DATA_BLOCK "DB2040_WINCC_HMI_LINES"   // DB2040
{ S7_Optimized_Access := 'FALSE'; DB_Accessible_From_OPC_UA := 'FALSE' }
AUTHOR : ETXETAR
VERSION : 1.0
// stored: AutoNumber false, DBAccessibleFromOPCUA false, DBAccessibleFromWebserver true, IsOnlyStoredInLoadMemory false, IsWriteProtectedInAS false
   VAR RETAIN
      MODES { S7_SetPoint := 'True'} : Array[1..5] of "WINCC_HMI_LINES";
      SERVICES { S7_SetPoint := 'True'} : Array[1..30] of "WINCC_HMI_LINES";
   END_VAR
BEGIN
   // MODES[1] : AUTOMATIC MODE
   // MODES[2] : SEMIAUTO MODE
   // MODES[3] : MANUAL MODE
   // MODES[1].WINCC_LINE_REQUEST_RIGHT : AUTOMATIC MODE RIGHT REQUEST
   // MODES[2].WINCC_LINE_REQUEST_RIGHT : SEMIAUTO MODE RIGHT REQUEST
   // MODES[3].WINCC_LINE_REQUEST_RIGHT : MANUAL MODE RIGHT REQUEST
   // MODES[1].WINCC_LINE_REQUEST_LEFT : AUTOMATIC MODE LEFT REQUEST
   // MODES[2].WINCC_LINE_REQUEST_LEFT : SEMIAUTO MODE LEFT REQUEST
   // MODES[3].WINCC_LINE_REQUEST_LEFT : MANUAL MODE LEFT REQUEST
   // MODES[1].WINCC_LINE_CONDITIONS_RIGHT : AUTOMATIC MODE RIGHT CONDITIONS
   // MODES[2].WINCC_LINE_CONDITIONS_RIGHT : SEMIAUTO MODE RIGHT CONDITIONS
   // MODES[3].WINCC_LINE_CONDITIONS_RIGHT : MANUAL MODE RIGHT CONDITIONS
   // MODES[1].WINCC_LINE_CONDITIONS_LEFT : AUTOMATIC MODE LEFT CONDITIONS
   // MODES[2].WINCC_LINE_CONDITIONS_LEFT : SEMIAUTO MODE LEFT CONDITIONS
   // MODES[3].WINCC_LINE_CONDITIONS_LEFT : MANUAL MODE LEFT CONDITIONS
   // MODES[1].WINCC_LINE_ACTIVE_RIGHT : AUTOMATIC MODE RIGHT ACTIVE
   // MODES[2].WINCC_LINE_ACTIVE_RIGHT : SEMIAUTO MODE RIGHT ACTIVE
   // MODES[3].WINCC_LINE_ACTIVE_RIGHT : MANUAL MODE RIGHT ACTIVE
   // MODES[1].WINCC_LINE_ACTIVE_LEFT : AUTOMATIC MODE LEFT ACTIVE
   // MODES[2].WINCC_LINE_ACTIVE_LEFT : SEMIAUTO MODE LEFT ACTIVE
   // MODES[3].WINCC_LINE_ACTIVE_LEFT : MANUAL MODE LEFT ACTIVE
   // MODES[1].WINCC_LINE_STATUS_1_RIGHT : AUTOMATIC MODE RIGHT STATUS
   // MODES[2].WINCC_LINE_STATUS_1_RIGHT : SEMIAUTO MODE RIGHT STATUS
   // MODES[3].WINCC_LINE_STATUS_1_RIGHT : MANUAL MODE RIGHT STATUS
   // MODES[1].WINCC_LINE_STATUS_1_LEFT : AUTOMATIC MODE LEFT STATUS
   // MODES[2].WINCC_LINE_STATUS_1_LEFT : SEMIAUTO MODE LEFT STATUS
   // MODES[3].WINCC_LINE_STATUS_1_LEFT : MANUAL MODE LEFT STATUS
   // SERVICES[1] : PNEUMATIC SYSTEM
   // SERVICES[2] : POWDER FEEDER 1 GENERAL UNIT 01
   // SERVICES[3] : POWDER FEEDER 1 GENERAL UNIT 02
   // SERVICES[4] : POWDER FEEDER 2 GENERAL UNIT 02
   // SERVICES[5] : POWDER FEEDER 1 HEATER JKL UNIT 01 LINE 1
   // SERVICES[6] : POWDER FEEDER 1 HEATER JKL UNIT 01 LINE 2
   // SERVICES[7] : POWDER FEEDER 1 HEATER JKL UNIT 02 LINE 1
   // SERVICES[8] : POWDER FEEDER 1 HEATER JKL UNIT 02 LINE 2
   // SERVICES[9] : POWDER FEEDER 2 HEATER JKL UNIT 02 LINE 1
   // SERVICES[10] : POWDER FEEDER 1 HOPPER UNIT 01 LINE 1
   // SERVICES[11] : POWDER FEEDER 1 HOPPER UNIT 01 LINE 2
   // SERVICES[12] : POWDER FEEDER 1 HOPPER UNIT 02 LINE 1
   // SERVICES[13] : POWDER FEEDER 1 HOPPER UNIT 02 LINE 2
   // SERVICES[14] : POWDER FEEDER 2 HOPPER UNIT 02 LINE 1
END_DATA_BLOCK

DATA_BLOCK "DB2041_WINCC_HMI_LINES_STATIONS"   // DB2041
{ S7_Optimized_Access := 'FALSE'; DB_Accessible_From_OPC_UA := 'FALSE' }
AUTHOR : ETXETAR
VERSION : 1.0
// stored: AutoNumber false, DBAccessibleFromOPCUA false, DBAccessibleFromWebserver true, IsOnlyStoredInLoadMemory false, IsWriteProtectedInAS false
   VAR RETAIN
      STATION_1 { S7_SetPoint := 'True'} : Array[1..20] of "WINCC_HMI_LINES";
      STATION_2 { S7_SetPoint := 'True'} : Array[1..20] of "WINCC_HMI_LINES";
      STATION_3 { S7_SetPoint := 'True'} : Array[1..20] of "WINCC_HMI_LINES";
      STATION_4 { S7_SetPoint := 'True'} : Array[1..20] of "WINCC_HMI_LINES";
      STATION_5 { S7_SetPoint := 'True'} : Array[1..20] of "WINCC_HMI_LINES";
      STATION_6 { S7_SetPoint := 'True'} : Array[1..20] of "WINCC_HMI_LINES";
      STATION_7 { S7_SetPoint := 'True'} : Array[1..20] of "WINCC_HMI_LINES";
      STATION_8 { S7_SetPoint := 'True'} : Array[1..20] of "WINCC_HMI_LINES";
      STATION_9 { S7_SetPoint := 'True'} : Array[1..20] of "WINCC_HMI_LINES";
      STATION_10 { S7_SetPoint := 'True'} : Array[1..20] of "WINCC_HMI_LINES";
   END_VAR
BEGIN
END_DATA_BLOCK

DATA_BLOCK "DB2050_HARDWARE_SOFTWARE_ENABLE_DISABLE"   // DB2050
{ S7_Optimized_Access := 'FALSE'; DB_Accessible_From_OPC_UA := 'FALSE' }
AUTHOR : ETXETAR
VERSION : 1.0
// stored: AutoNumber false, DBAccessibleFromOPCUA false, DBAccessibleFromWebserver true, IsOnlyStoredInLoadMemory false, IsWriteProtectedInAS false
   VAR RETAIN
      DISABLE_PART : Struct
         HW_GENERAL_CONDITIONS : Bool;   // HARDWARE GENERAL CONDITIONS
         SW_GENERAL_CONDITIONS : Bool;   // SOFTWARE GENERAL CONDITIONS
         PART_A_ENABLE : Bool;   // PART A ENABLE
         PART_B_ENABLE : Bool;   // PART B ENABLE
         PART_C_ENABLE : Bool;   // PART C ENABLE
         PART_D_ENABLE : Bool;   // PART D ENABLE
         PART_E_ENABLE : Bool;   // PART E ENABLE
         PART_F_ENABLE : Bool;   // PART F ENABLE
         HW_PART_A_ENABLE_REQUEST : Bool;   // HARDWARE PART A ENABLE REQUEST
         HW_PART_A_DISABLE_REQUEST : Bool;   // HARDWARE PART A DISABLE REQUEST
         HW_PART_B_ENABLE_REQUEST : Bool;   // HARDWARE PART B ENABLE REQUEST
         HW_PART_B_DISABLE_REQUEST : Bool;   // HARDWARE PART B DISABLE REQUEST
         HW_PART_C_ENABLE_REQUEST : Bool;   // HARDWARE PART C ENABLE REQUEST
         HW_PART_C_DISABLE_REQUEST : Bool;   // HARDWARE PART C DISABLE REQUEST
         HW_PART_D_ENABLE_REQUEST : Bool;   // HARDWARE PART D ENABLE REQUEST
         HW_PART_D_DISABLE_REQUEST : Bool;   // HARDWARE PART D DISABLE REQUEST
         HW_PART_E_ENABLE_REQUEST : Bool;   // HARDWARE PART E ENABLE REQUEST
         HW_PART_E_DISABLE_REQUEST : Bool;   // HARDWARE PART E DISABLE REQUEST
         HW_PART_F_ENABLE_REQUEST : Bool;   // HARDWARE PART F ENABLE REQUEST
         HW_PART_F_DISABLE_REQUEST : Bool;   // HARDWARE PART F DISABLE REQUEST
         HW_PART_ENABLE_DISABLE_REQUEST : Bool;   // HARDWARE ENABLE DISABLE REQUEST
         SW_PART_A_ENABLE_REQUEST : Bool;   // SOFTWARE PART A ENABLE REQUEST
         SW_PART_A_DISABLE_REQUEST : Bool;   // SOFTWARE PART A DISABLE REQUEST
         SW_PART_B_ENABLE_REQUEST : Bool;   // SOFTWARE PART B ENABLE REQUEST
         SW_PART_B_DISABLE_REQUEST : Bool;   // SOFTWARE PART B DISABLE REQUEST
         SW_PART_C_ENABLE_REQUEST : Bool;   // SOFTWARE PART C ENABLE REQUEST
         SW_PART_C_DISABLE_REQUEST : Bool;   // SOFTWARE PART C DISABLE REQUEST
         SW_PART_D_ENABLE_REQUEST : Bool;   // SOFTWARE PART D ENABLE REQUEST
         SW_PART_D_DISABLE_REQUEST : Bool;   // SOFTWARE PART D DISABLE REQUEST
         SW_PART_E_ENABLE_REQUEST : Bool;   // SOFTWARE PART E ENABLE REQUEST
         SW_PART_E_DISABLE_REQUEST : Bool;   // SOFTWARE PART E DISABLE REQUEST
         SW_PART_F_ENABLE_REQUEST : Bool;   // SOFTWARE PART F ENABLE REQUEST
         SW_PART_F_DISABLE_REQUEST : Bool;   // SOFTWARE PART F DISABLE REQUEST
         SW_PART_ENABLE_DISABLE_REQUEST : Bool;   // SOFTWARE ENABLE DISABLE REQUEST
         HMI_ACCEPT_BUTTON : Bool;   // HMI ACCEPT BUTTON
         HW_PART_A_ENABLED : Bool := true;   // HARDWARE PART A ENABLED
         HW_PART_B_ENABLED : Bool := true;   // HARDWARE PART B ENABLED
         HW_PART_C_ENABLED : Bool := true;   // HARDWARE PART C ENABLED
         HW_PART_D_ENABLED : Bool;   // HARDWARE PART D ENABLED
         HW_PART_E_ENABLED : Bool;   // HARDWARE PART E ENABLED
         HW_PART_F_ENABLED : Bool;   // HARDWARE PART F ENABLED
         SW_PART_A_ENABLED : Bool := true;   // SOFTWARE PART A ENABLED
         SW_PART_B_ENABLED : Bool := true;   // SOFTWARE PART B ENABLED
         SW_PART_C_ENABLED : Bool := true;   // SOFTWARE PART C ENABLED
         SW_PART_D_ENABLED : Bool;   // SOFTWARE PART D ENABLED
         SW_PART_E_ENABLED : Bool;   // SOFTWARE PART E ENABLED
         SW_PART_F_ENABLED : Bool;   // SOFTWARE PART F ENABLED
         PART_A_DISABLE_ALARM : Bool;   // PART A DISABLE ALARM
         PART_B_DISABLE_ALARM : Bool;   // PART B DISABLE ALARM
         PART_C_DISABLE_ALARM : Bool;   // PART C DISABLE ALARM
         PART_D_DISABLE_ALARM : Bool;   // PART D DISABLE ALARM
         PART_E_DISABLE_ALARM : Bool;   // PART E DISABLE ALARM
         PART_F_DISABLE_ALARM : Bool;   // PART F DISABLE ALARM
         DESELECT_IN_PROGRESS : Bool;   // DESELECTION IN PROGRESS
         HW_DISABLED_ACK : Bool;   // HARDWARE DISABLED ACKNOWLEDGE
         HW_DISABLED_ACK_AUX : Bool;   // HARDWARE DISABLED ACKNOWLEDGE AUXILIARY
         ALL_HW_PARTS_DISABLED : Bool;   // ALL HARDWARE PARTS DISABLED
         ALL_SW_PARTS_DISABLED : Bool;   // ALL SOFTWARE PARTS DISABLED
         ALL_HARDWARE_ENABLED : Bool;   // ALL HARDWARE ENABLED
         PART_A_DISABLED_SCRIPT_COMMAND : Bool;   // PART A DISABLED SCRIPT COMMAND
         PART_A_ENABLED_SCRIPT_COMMAND : Bool;   // PART A ENABLED SCRIPT COMMAND
         PART_B_DISABLED_SCRIPT_COMMAND : Bool;   // PART B DISABLED SCRIPT COMMAND
         PART_B_ENABLED_SCRIPT_COMMAND : Bool;   // PART B ENABLED SCRIPT COMMAND
         PART_C_DISABLED_SCRIPT_COMMAND : Bool;   // PART C DISABLED SCRIPT COMMAND
         PART_C_ENABLED_SCRIPT_COMMAND : Bool;   // PART C ENABLED SCRIPT COMMAND
         PART_D_DISABLED_SCRIPT_COMMAND : Bool;   // PART D DISABLED SCRIPT COMMAND
         PART_D_ENABLED_SCRIPT_COMMAND : Bool;   // PART D ENABLED SCRIPT COMMAND
         PART_E_DISABLED_SCRIPT_COMMAND : Bool;   // PART E DISABLED SCRIPT COMMAND
         PART_E_ENABLED_SCRIPT_COMMAND : Bool;   // PART E ENABLED SCRIPT COMMAND
         PART_F_DISABLED_SCRIPT_COMMAND : Bool;   // PART F DISABLED SCRIPT COMMAND
         PART_F_ENABLED_SCRIPT_COMMAND : Bool;   // PART F ENABLED SCRIPT COMMAND
         ALARM_SCREEN : Int;   // HMI ALARMS SCREEN NUMBER
         ENABLE_MACHINE_STRUCTURE_SCREEN : Int;   // HMI ENABLE MACHINE STRUCTURE SCREEN NUMBER
         SW_PULSE : Array[1..16] of Bool;
         HW_PULSE : Array[1..16] of Bool;
      END_STRUCT;
   END_VAR
BEGIN
END_DATA_BLOCK

DATA_BLOCK "DB21000_POWDER_FEEDER_GENERAL"   // DB21000
{ S7_Optimized_Access := 'FALSE'; DB_Accessible_From_OPC_UA := 'FALSE' }
VERSION : 0.1
// stored: AutoNumber false, DBAccessibleFromOPCUA false, DBAccessibleFromWebserver true, IsOnlyStoredInLoadMemory false, IsWriteProtectedInAS false
   VAR
      POWDER_FEEDER_1_UNIT_01 : "POWDER FEEDER GENERAL";
      POWDER_FEEDER_1_UNIT_02 { S7_SetPoint := 'True'} : "POWDER FEEDER GENERAL";
      POWDER_FEEDER_2_UNIT_02 { S7_SetPoint := 'True'} : "POWDER FEEDER GENERAL";
   END_VAR
BEGIN
END_DATA_BLOCK

DATA_BLOCK "DB21002_POWDER_FEEDER_OERLIKON_INTERLOCK"   // DB21002
{ S7_Optimized_Access := 'FALSE'; DB_Accessible_From_OPC_UA := 'FALSE' }
VERSION : 0.1
// stored: AutoNumber false, DBAccessibleFromOPCUA false, DBAccessibleFromWebserver true, IsOnlyStoredInLoadMemory false, IsWriteProtectedInAS false
   VAR
      POWDER_FEEDER_1_UNIT_01 : "POWDER FEEDER OERLIKON";
      POWDER_FEEDER_1_UNIT_02 : "POWDER FEEDER OERLIKON";
      POWDER_FEEDER_2_UNIT_02 : "POWDER FEEDER OERLIKON";
   END_VAR
BEGIN
END_DATA_BLOCK

DATA_BLOCK "DB21003_POWDER_FEEDER_HMI_INTERLOCK"   // DB21003
{ S7_Optimized_Access := 'FALSE'; DB_Accessible_From_OPC_UA := 'FALSE' }
VERSION : 0.1
// stored: AutoNumber false, DBAccessibleFromOPCUA false, DBAccessibleFromWebserver true, IsOnlyStoredInLoadMemory false, IsWriteProtectedInAS false
   VAR
      POWDER_FEEDER_1_UNIT_01 : Struct
         "HMI_Values Setpoints" : "POWDER FEEDER HMI VALUES SETPOINTS";
         "HMI_Offsets Alarms and Warnings" : "POWDER FEEDER HMI OFFSETS ALARMS WARNINGS";
         HMI_ACTIONS_STATUS { S7_SetPoint := 'True'} : "POWDER FEEDER HMI ACTIONS";
      END_STRUCT;
      POWDER_FEEDER_1_UNIT_02 : Struct
         "HMI_Values Setpoints" : "POWDER FEEDER HMI VALUES SETPOINTS";
         "HMI_Offsets Alarms and Warnings" : "POWDER FEEDER HMI OFFSETS ALARMS WARNINGS";
         HMI_ACTIONS_STATUS : "POWDER FEEDER HMI ACTIONS";
      END_STRUCT;
      POWDER_FEEDER_2_UNIT_02 : Struct
         "HMI_Values Setpoints" : "POWDER FEEDER HMI VALUES SETPOINTS";
         "HMI_Offsets Alarms and Warnings" : "POWDER FEEDER HMI OFFSETS ALARMS WARNINGS";
         HMI_ACTIONS_STATUS : "POWDER FEEDER HMI ACTIONS";
      END_STRUCT;
   END_VAR
BEGIN
END_DATA_BLOCK

DATA_BLOCK "DB21004_POWDER_FEEDER_CNC_INTERLOCK"   // DB21004
{ S7_Optimized_Access := 'FALSE'; DB_Accessible_From_OPC_UA := 'FALSE' }
VERSION : 0.1
// stored: AutoNumber false, DBAccessibleFromOPCUA false, DBAccessibleFromWebserver true, IsOnlyStoredInLoadMemory false, IsWriteProtectedInAS false
   VAR
      POWDER_FEEDER_1_UNIT_01 : "POWDER FEEDER CNC VALUES SETPOINTS";
      POWDER_FEEDER_1_UNIT_02 : "POWDER FEEDER CNC VALUES SETPOINTS";
      POWDER_FEEDER_2_UNIT_02 : "POWDER FEEDER CNC VALUES SETPOINTS";
   END_VAR
BEGIN
END_DATA_BLOCK

DATA_BLOCK "DB21005_POWDER_FEEDER_PLC_AUX"   // DB21005
{ S7_Optimized_Access := 'FALSE'; DB_Accessible_From_OPC_UA := 'FALSE' }
VERSION : 0.1
// stored: AutoNumber false, DBAccessibleFromOPCUA false, DBAccessibleFromWebserver true, IsOnlyStoredInLoadMemory false, IsWriteProtectedInAS false
   VAR
      "INTERLOCKS_PLC_I/O_PF_1_UNIT_01" : "POWDER FEEDER PLC AUXILIAR";
      "INTERLOCKS_PLC_I/O_PF_1_UNIT_02" : "POWDER FEEDER PLC AUXILIAR";
      "INTERLOCKS_PLC_I/O_PF_2_UNIT_02" : "POWDER FEEDER PLC AUXILIAR";
   END_VAR
BEGIN
END_DATA_BLOCK

DATA_BLOCK "DB1101_MACHINE_SEQUENCE"   // DB1101
{ S7_Optimized_Access := 'FALSE'; DB_Accessible_From_OPC_UA := 'FALSE' }
AUTHOR : ETXETAR
VERSION : 1.0
// stored: AutoNumber false, DBAccessibleFromOPCUA false, DBAccessibleFromWebserver true, IsOnlyStoredInLoadMemory false, IsWriteProtectedInAS false
   VAR RETAIN
      GENERAL_CONDITIONS : Bool;   // MACHINING SEQUENCE GENERAL CONDITIONS / MACHINE SEQUENCE GENERAL CONDITIONS
      INITIAL_CONDITIONS : Bool;   // MACHINING SEQUENCE INITIAL CONDITIONS / MACHINE SEQUENCE INITIAL CONDITIONS
      START_REQUEST : Bool;   // MACHINING SEQUENCE START REQUEST / MACHINE SEQUENCE START REQUEST
      COMMAND : Bool;   // MACHINING SEQUENCE COMMAND / MACHINE SEQUENCE COMMAND
      REQUEST : Bool;   // MACHINING SEQUENCE REQUEST DELAYED / MACHINE SEQUENCE REQUEST
      COMMAND_PULSE : Bool;   // MACHINING SEQUENCE COMMAND PULSE / MACHINE SEQUENCE COMMAND PULSE
      REQUEST_PULSE : Bool;   // MACHINING SEQUENCE REQUEST PULSE / MACHINE SEQUENCE REQUEST PULSE
      RUNNING : Bool;   // MACHINING SEQUENCE IN PROCESS / MACHINE SEQUENCE RUNNING
      CYCLE_UNIT_01 : Bool;   // MACHINING SEQUENCE CYCLE STATION 01R / MACHINE SEQUENCE CYCLE UNIT 01
      CYCLE_UNIT_02 : Bool;   // MACHINING SEQUENCE CYCLE STATION 01L / MACHINE SEQUENCE CYCLE UNIT 02
      CYCLE_UNIT_03 : Bool;   // MACHINING SEQUENCE CYCLE STATION 01L / MACHINE SEQUENCE CYCLE UNIT 03
      NO_PART_AT_FEED_UNIT_01 : Bool;   // MACHINING SEQUENCE CYCLE STATION FIXTURE / MACHINE SEQUENCE NO PART AT FEED UNIT 02
      DELIVERY_OCCUPIED_UNIT_01 : Bool;   // MACHINING SEQUENCE CYCLE PART HANDLING DEVICE / MACHINE SEQUENCE DELIVERY OCCUPIED UNIT 02
      NO_PART_AT_FEED_UNIT_02 : Bool;   // MACHINING SEQUENCE NO PART AT FEED / MACHINE SEQUENCE NO PART AT FEED UNIT 02
      DELIVERY_OCCUPIED_UNIT_02 : Bool;   // MACHINING SEQUENCE DELIVERY OCCUPIED / MACHINE SEQUENCE DELIVERY OCCUPIED UNIT 02
      CLEAR_TO_LOAD_UNLOAD_UNIT_01 : Bool;   // MACHINING SEQUENCE OUT OF COLLISION TO PART HANDLING DEVICE / MACHINE SEQUENCE CLEAR TO LOAD UNLOAD MACHINE UNIT 01
      CLEAR_TO_LOAD_UNLOAD_UNIT_02 : Bool;   // MACHINING SEQUENCE OUT OF COLLISION TO PART HANDLING DEVICE / MACHINE SEQUENCE CLEAR TO LOAD UNLOAD MACHINE UNIT 02
      SKIP_FIXTURE_UNIT_01 : Bool;   // MACHINING SEQUENCE CLAMP FIXTURE 1 / MACHINE SEQUENCE SKIP FIXTURE UNIT 01
      SKIP_FIXTURE_UNIT_02 : Bool;   // MACHINING SEQUENCE CLAMP FIXTURE 2 / MACHINE SEQUENCE SKIP FIXTURE UNIT 02
      SPARE_1 : Bool;   // MACHINING SEQUENCE UNCLAMP FIXTURE 1 / MACHINE SEQUENCE
      SPARE_2 : Bool;   // MACHINING SEQUENCE UNCLAMP FIXTURE 2 / MACHINE SEQUENCE
      RESET_PLC_AND_CNC : Bool;   // MACHINING SEQUENCE RESET PLC AND CNC / MACHINE SEQUENCE RESET PLC AND CNC
      FULL_DEPTH : Bool;   // MACHINING SEQUENCE FULL DEPTH / MACHINE SEQUENCE FULL DEPTH
      TIME_EXCEEDED : Bool;   // MACHINING SEQUENCE TIME EXCEEDED / MACHINE SEQUENCE TIME EXCEEDED
      PREALARM : Bool;   // MACHINING SEQUENCE PREALARM / MACHINE SEQUENCE PREALARM
      LOADER_CHECK_PART_READY : Bool;   // MACHINING SEQUENCE LOADER CHECK PART READY / MACHINE SEQUENCE LOADER CHECK PART READY
      LOADER_RESET_CHECK_PART_READY : Bool;   // MACHINING SEQUENCE RST LOADER CHECK PART READY / MACHINE SEQUENCE LOADER RESET CHECK PART READY
      PREALARM_GONE : Bool;   // MACHINING SEQUENCE PREALARM GONE / MACHINE SEQUENCE PREALARM GONE
      AUX1 : Bool;   // MACHINING SEQUENCE AUX1 / MACHINE SEQUENCE AUX1
      AUX2 : Bool;   // MACHINING SEQUENCE AUX2 / MACHINE SEQUENCE AUX2
      AUX3 : Bool;   // MACHINING SEQUENCE AUX3 / MACHINE SEQUENCE AUX3
      START_GENERAL_COND_HELP : Bool;   // MACHINING SEQUENCE START GENERAL CONDITIONS HELP / MACHINE SEQUENCE START GENERAL COND HELP
      START_INITIAL_COND_HELP : Bool;   // MACHINING SEQUENCE START INITIAL CONDITIONS HELP / MACHINE SEQUENCE START INITIAL COND HELP
      TIMER_MACHINE_START_REQUEST : TON_TIME;   // MACHINE SEQUENCE START REQUEST TIMER
      "TIMER_TIME _EXCEEDED" : TON_TIME;   // MACHINE SEQUENCE TIME EXCEEDED TIMER
      TIMER_UNLOAD_UNIT_01_DELAY : TON_TIME;   // MACHINE SEQUENCE UNLOAD UNIT 01 DELAY TIMER
      TIMER_LOAD_UNIT_01_DELAY : TON_TIME;   // MACHINE SEQUENCE LOAD UNIT 01 DELAY TIMER
      TIMER_UNLOAD_UNIT_02_DELAY : TON_TIME;   // MACHINE SEQUENCE UNLOAD UNIT 02 DELAY TIMER
      TIMER_LOAD_UNIT_02_DELAY : TON_TIME;   // MACHINE SEQUENCE LOAD UNIT 02 DELAY TIMER
   END_VAR
BEGIN
   TIMER_MACHINE_START_REQUEST.PT := T#3s;
   "TIMER_TIME _EXCEEDED".PT := T#800s;
   TIMER_UNLOAD_UNIT_01_DELAY.PT := T#500ms;
   TIMER_LOAD_UNIT_01_DELAY.PT := T#1s;
   TIMER_UNLOAD_UNIT_02_DELAY.PT := T#500ms;
   TIMER_LOAD_UNIT_02_DELAY.PT := T#1s;
END_DATA_BLOCK

DATA_BLOCK "DB2001_MODES_GENERAL"   // DB2001
{ S7_Optimized_Access := 'FALSE'; DB_Accessible_From_OPC_UA := 'FALSE' }
AUTHOR : ETXETAR
VERSION : 1.0
// stored: AutoNumber false, DBAccessibleFromOPCUA false, DBAccessibleFromWebserver true, IsOnlyStoredInLoadMemory false, IsWriteProtectedInAS false
   VAR RETAIN
      GENERAL : "AUTO_SINGLE_SEMI_MANUAL";
      STEP_BY_STEP { S7_SetPoint := 'True'} : "MODES";
      MDA { S7_SetPoint := 'True'} : "MODES";
      REFERENCE { S7_SetPoint := 'True'} : "MODES";
      INCREMENTAL { S7_SetPoint := 'True'} : "INCREMENTAL";
      BA { S7_SetPoint := 'True'} : "BA_MODE";
   END_VAR
BEGIN
   // STEP_BY_STEP.MODE_SELECTED : STEP BY STEP MODE SELECTED
   // MDA.MODE_SELECTED : MDA MODE SELECTED
   // REFERENCE.MODE_SELECTED : REFERENCE MODE SELECTED
END_DATA_BLOCK

DATA_BLOCK "DB2011_MODES_GENERAL_MG2"   // DB2011
{ S7_Optimized_Access := 'FALSE'; DB_Accessible_From_OPC_UA := 'FALSE' }
AUTHOR : ETXETAR
VERSION : 1.0
// stored: AutoNumber false, DBAccessibleFromOPCUA false, DBAccessibleFromWebserver true, IsOnlyStoredInLoadMemory false, IsWriteProtectedInAS false
   VAR RETAIN
      GENERAL : "AUTO_SINGLE_SEMI_MANUAL";
      STEP_BY_STEP { S7_SetPoint := 'True'} : "MODES";
      MDA { S7_SetPoint := 'True'} : "MODES";
      REFERENCE { S7_SetPoint := 'True'} : "MODES";
      INCREMENTAL { S7_SetPoint := 'True'} : "INCREMENTAL";
      BA { S7_SetPoint := 'True'} : "BA_MODE";
   END_VAR
BEGIN
   // STEP_BY_STEP.MODE_SELECTED : STEP BY STEP MODE SELECTED
   // MDA.MODE_SELECTED : MDA MODE SELECTED
   // REFERENCE.MODE_SELECTED : REFERENCE MODE SELECTED
END_DATA_BLOCK

DATA_BLOCK "DB2099_MANUAL_LOAD_DMC"   // DB2099
{ S7_Optimized_Access := 'FALSE'; DB_Accessible_From_OPC_UA := 'FALSE' }
VERSION : 0.1
// stored: AutoNumber false, DBAccessibleFromOPCUA false, DBAccessibleFromWebserver true, IsOnlyStoredInLoadMemory false, IsWriteProtectedInAS false
   VAR
      DMC_UNIT_01_HMI : Array[0..99] of Char;   // DMC UNIT 01 IN THE HMI
      DMC_UNIT_02_HMI : Array[0..99] of Char;   // DMC UNIT 02 IN THE HMI
      DMC_STRING_UNIT_01 : String;   // DMC AUX STRING UNIT 01
      DMC_STRING_UNIT_02 : String;   // DMC AUX STRING UNIT 02
      AUX_CNT_INT_UNIT_01 : Int;
      AUX_CNT_INT_UNIT_02 : Int;
      DMC_ARRAY_CHAR_UNIT_01 : Array[0..99] of Char;   // DMC ARRAY UNIT 01
      DMC_ARRAY_CHAR_UNIT_02 : Array[0..99] of Char;   // DMC ARRAY UNIT 02
      MANUAL_LOADING_OR_DRY_PART_LOADED_UNIT_01 : Bool;   // MANUAL LOADING OR DRY CYCLE PART LOADED IN UNIT 01
      MANUAL_LOADING_OR_DRY_PART_LOADED_UNIT_02 : Bool;   // MANUAL LOADING OR DRY CYCLE PART LOADED IN UNIT 02
      MANUAL_LOADING_OR_DRY_PART_UNLOADED_UNIT_01 : Bool;   // MANUAL LOADING OR DRY CYCLE PART UNLOADED IN UNIT 01
      MANUAL_LOADING_OR_DRY_PART_UNLOADED_UNIT_02 : Bool;   // MANUAL LOADING OR DRY CYCLE PART UNLOADED IN UNIT 02
      MANUAL_LOADING_OR_DRY_PART_LOADED_UNIT_01_P : Bool;   // MANUAL LOADING OR DRY CYCLE PART LOADED IN UNIT 01 PULSE
      MANUAL_LOADING_OR_DRY_PART_LOADED_UNIT_02_P : Bool;   // MANUAL LOADING OR DRY CYCLE PART LOADED IN UNIT 02 PULSE
      MANUAL_LOADING_OR_DRY_PART_UNLOADED_UNIT_01_P : Bool;   // MANUAL LOADING OR DRY CYCLE PART UNLOADED IN UNIT 01 PULSE
      MANUAL_LOADING_OR_DRY_PART_UNLOADED_UNIT_02_P : Bool;   // MANUAL LOADING OR DRY CYCLE PART UNLOADED IN UNIT 02 PULSE
      START_DMC_NUMBER_INT : DInt;
      START_DMC_NUMBER_STRING : String;
      START_DMC_NUMBER_CHAR_ARRAY : Array[0..10] of Char;
      AUX_CNT_START_DMC_NUMBER : Int;
      PULSE_1 : Bool;
      PRODUCTION_SELECTED : Bool;
   END_VAR
BEGIN
END_DATA_BLOCK

DATA_BLOCK "DB2109_STATION_3_LIGHT_U01"   // DB2109
{ S7_Optimized_Access := 'FALSE'; DB_Accessible_From_OPC_UA := 'FALSE' }
AUTHOR : ETXETAR
VERSION : 1.0
// stored: AutoNumber false, DBAccessibleFromOPCUA false, DBAccessibleFromWebserver true, IsOnlyStoredInLoadMemory false, IsWriteProtectedInAS false
   VAR RETAIN
      I_CIRCUIT_BREAKER : Bool;   // CIRCUIT BREAKER INPUT
      I_SELECTOR_ON : Bool;   // SELECTOR ON INPUT
      SWITCH_ON_GENERAL_CONDITIONS : Bool;   // SWITCH ON GENERAL CONDITIONS
      SWITCH_ON_INITIAL_CONDITIONS : Bool;   // SWITCH ON INITIAL CONDITIONS
      SWITCH_ON_MANUAL_REQUEST : Bool;   // SWITCH ON MANUAL REQUEST
      SWITCH_ON_AUTO_REQUEST : Bool;   // SWITCH ON AUTO REQUEST
      SWITCH_ON_GLOBAL_REQUEST : Bool;   // SWITCH ON GLOBAL REQUEST
      SWITCH_ON_COMMAND : Bool;   // SWITCH ON COMMAND
      SWITCH_ON : Bool;   // SWITCH ON
      IN_SERVICE : Bool;   // IN SERVICE
      SWITCH_OFF_GENERAL_CONDITIONS : Bool;   // SWITCH OFF GENERAL CONDITIONS
      SWITCH_OFF_INITIAL_CONDITIONS : Bool;   // SWITCH OFF INITIAL CONDITIONS
      SWITCH_OFF_MANUAL_REQUEST : Bool;   // SWITCH OFF MANUAL REQUEST
      SWITCH_OFF_AUTO_REQUEST : Bool;   // SWITCH OFF AUTO REQUEST
      SWITCH_OFF_GLOBAL_REQUEST : Bool;   // SWITCH OFF GLOBAL REQUEST
      SWITCH_OFF_COMMAND : Bool;   // SWITCH OFF COMMAND
      SWITCH_OFF : Bool;   // SWITCH OFF
      OUT_OF_SERVICE : Bool;   // OUT OF SERVICE
      SWITCH_ON_GENERAL_CONDITIONS_HELP : Bool;   // SWITCH ON GENERAL CONDITIONS HELP
      SWITCH_ON_INITIAL_CONDITIONS_HELP : Bool;   // SWITCH ON INITIAL CONDITIONS HELP
      SWITCH_OFF_GENERAL_CONDITIONS_HELP : Bool;   // SWITCH OFF GENERAL CONDITIONS HELP
      SWITCH_OFF_INITIAL_CONDITIONS_HELP : Bool;   // SWITCH OFF INITIAL CONDITIONS HELP
      SWITCH_ON_GLOBAL_REQUEST_AUX1 : Bool;   // SWITCH ON GLOBAL REQUEST ON AUXILIARY 1
      SWITCH_ON_GLOBAL_REQUEST_AUX2 : Bool;   // SWITCH ON GLOBAL REQUEST ON AUXILIARY 2
      SWITCH_ON_GLOBAL_REQUEST_AUX3 : Bool;   // SWITCH ON GLOBAL REQUEST ON AUXILIARY 3
      SWITCH_OFF_AUTO_REQUEST_AUX : Bool;   // INITIAL AUX 4
      SWITCH_OFF_GLOBAL_REQUEST_AUX : Bool;   // INITIAL AUX 5
      TIMER_SWITCH_OFF_1 : TON_TIME;   // SWITCH OFF GLOBAL REQUEST 1 TIMER
      TIMER_SWITCH_OFF_2 : TON_TIME;   // SWITCH OFF GLOBAL REQUEST 2 TIMER
   END_VAR
BEGIN
   TIMER_SWITCH_OFF_1.PT := T#10M;
   TIMER_SWITCH_OFF_2.PT := T#1H;
END_DATA_BLOCK

DATA_BLOCK "DB2110_STATION_3_LIGHT_U02"   // DB2110
{ S7_Optimized_Access := 'FALSE'; DB_Accessible_From_OPC_UA := 'FALSE' }
AUTHOR : ETXETAR
VERSION : 1.0
// stored: AutoNumber false, DBAccessibleFromOPCUA false, DBAccessibleFromWebserver true, IsOnlyStoredInLoadMemory false, IsWriteProtectedInAS false
   VAR RETAIN
      I_CIRCUIT_BREAKER : Bool;   // CIRCUIT BREAKER INPUT
      I_SELECTOR_ON : Bool;   // SELECTOR ON INPUT
      SWITCH_ON_GENERAL_CONDITIONS : Bool;   // SWITCH ON GENERAL CONDITIONS
      SWITCH_ON_INITIAL_CONDITIONS : Bool;   // SWITCH ON INITIAL CONDITIONS
      SWITCH_ON_MANUAL_REQUEST : Bool;   // SWITCH ON MANUAL REQUEST
      SWITCH_ON_AUTO_REQUEST : Bool;   // SWITCH ON AUTO REQUEST
      SWITCH_ON_GLOBAL_REQUEST : Bool;   // SWITCH ON GLOBAL REQUEST
      SWITCH_ON_COMMAND : Bool;   // SWITCH ON COMMAND
      SWITCH_ON : Bool;   // SWITCH ON
      IN_SERVICE : Bool;   // IN SERVICE
      SWITCH_OFF_GENERAL_CONDITIONS : Bool;   // SWITCH OFF GENERAL CONDITIONS
      SWITCH_OFF_INITIAL_CONDITIONS : Bool;   // SWITCH OFF INITIAL CONDITIONS
      SWITCH_OFF_MANUAL_REQUEST : Bool;   // SWITCH OFF MANUAL REQUEST
      SWITCH_OFF_AUTO_REQUEST : Bool;   // SWITCH OFF AUTO REQUEST
      SWITCH_OFF_GLOBAL_REQUEST : Bool;   // SWITCH OFF GLOBAL REQUEST
      SWITCH_OFF_COMMAND : Bool;   // SWITCH OFF COMMAND
      SWITCH_OFF : Bool;   // SWITCH OFF
      OUT_OF_SERVICE : Bool;   // OUT OF SERVICE
      SWITCH_ON_GENERAL_CONDITIONS_HELP : Bool;   // SWITCH ON GENERAL CONDITIONS HELP
      SWITCH_ON_INITIAL_CONDITIONS_HELP : Bool;   // SWITCH ON INITIAL CONDITIONS HELP
      SWITCH_OFF_GENERAL_CONDITIONS_HELP : Bool;   // SWITCH OFF GENERAL CONDITIONS HELP
      SWITCH_OFF_INITIAL_CONDITIONS_HELP : Bool;   // SWITCH OFF INITIAL CONDITIONS HELP
      SWITCH_ON_GLOBAL_REQUEST_AUX1 : Bool;   // SWITCH ON GLOBAL REQUEST ON AUXILIARY 1
      SWITCH_ON_GLOBAL_REQUEST_AUX2 : Bool;   // SWITCH ON GLOBAL REQUEST ON AUXILIARY 2
      SWITCH_ON_GLOBAL_REQUEST_AUX3 : Bool;   // SWITCH ON GLOBAL REQUEST ON AUXILIARY 3
      SWITCH_OFF_AUTO_REQUEST_AUX : Bool;   // INITIAL AUX 4
      SWITCH_OFF_GLOBAL_REQUEST_AUX : Bool;   // INITIAL AUX 5
      TIMER_SWITCH_OFF_1 : TON_TIME;   // SWITCH OFF GLOBAL REQUEST 1 TIMER
      TIMER_SWITCH_OFF_2 : TON_TIME;   // SWITCH OFF GLOBAL REQUEST 2 TIMER
   END_VAR
BEGIN
   TIMER_SWITCH_OFF_1.PT := T#10M;
   TIMER_SWITCH_OFF_2.PT := T#1H;
END_DATA_BLOCK

DATA_BLOCK "DB2500_UNIT_01_FIXTURE_1"   // DB2500
{ S7_Optimized_Access := 'FALSE'; DB_Accessible_From_OPC_UA := 'FALSE' }
AUTHOR : ETXETAR
VERSION : 1.0
// stored: AutoNumber false, DBAccessibleFromOPCUA false, DBAccessibleFromWebserver true, IsOnlyStoredInLoadMemory false, IsWriteProtectedInAS false
   VAR RETAIN
      INPUT_PART_A_PRESENT : Bool;   // UNIT 01 UNIT 01 FIXTURE 1 INPUT PART A PRESENT
      INPUT_PART_B_PRESENT : Bool;   // UNIT 01 FIXTURE 1 INPUT PART B PRESENT
      INPUT_PART_C_PRESENT : Bool;   // UNIT 01 FIXTURE 1 INPUT PART C PRESENT
      INPUT_PART_D_PRESENT : Bool;   // UNIT 01 FIXTURE 1 INPUT PART D PRESENT
      INPUT_PART_A_PRESENT_FACE_N : Bool;   // UNIT 01 FIXTURE 1 INPUT PART A PRESENT FACE N UP
      INPUT_PART_B_PRESENT_FACE_N : Bool;   // UNIT 01 FIXTURE 1 INPUT PART B PRESENT FACE N UP
      INPUT_PART_C_PRESENT_FACE_N : Bool;   // UNIT 01 FIXTURE 1 INPUT PART C PRESENT FACE N UP
      INPUT_PART_D_PRESENT_FACE_N : Bool;   // UNIT 01 FIXTURE 1 INPUT PART D PRESENT FACE N UP
      INPUT_PART_A_PRESENT_FACE_R : Bool;   // UNIT 01 FIXTURE 1 INPUT PART A PRESENT FACE R UP
      INPUT_PART_B_PRESENT_FACE_R : Bool;   // UNIT 01 FIXTURE 1 INPUT PART B PRESENT FACE R UP
      INPUT_PART_C_PRESENT_FACE_R : Bool;   // UNIT 01 FIXTURE 1 INPUT PART C PRESENT FACE R UP
      INPUT_PART_D_PRESENT_FACE_R : Bool;   // UNIT 01 FIXTURE 1 INPUT PART D PRESENT FACE R UP
      INPUT_PART_A_PRESENT_MEM : Bool;   // UNIT 01 FIXTURE 1 INPUT PART A PRESENT MEMORY
      INPUT_PART_B_PRESENT_MEM : Bool;   // UNIT 01 FIXTURE 1 INPUT PART B PRESENT MEMORY
      INPUT_PART_C_PRESENT_MEM : Bool;   // UNIT 01 FIXTURE 1 INPUT PART C PRESENT MEMORY
      INPUT_PART_D_PRESENT_MEM : Bool;   // UNIT 01 FIXTURE 1 INPUT PART D PRESENT MEMORY
      INPUT_PART_A_PRESENT_FACE_N_MEM : Bool;   // UNIT 01 FIXTURE 1 INPUT PART A PRESENT FACE N UP MEMORY
      INPUT_PART_B_PRESENT_FACE_N_MEM : Bool;   // UNIT 01 FIXTURE 1 INPUT PART B PRESENT FACE N UP MEMORY
      INPUT_PART_C_PRESENT_FACE_N_MEM : Bool;   // UNIT 01 FIXTURE 1 INPUT PART C PRESENT FACE N UP MEMORY
      INPUT_PART_D_PRESENT_FACE_N_MEM : Bool;   // UNIT 01 FIXTURE 1 INPUT PART D PRESENT FACE N UP MEMORY
      INPUT_PART_A_PRESENT_FACE_R_MEM : Bool;   // UNIT 01 FIXTURE 1 INPUT PART A PRESENT FACE R UP MEMORY
      INPUT_PART_B_PRESENT_FACE_R_MEM : Bool;   // UNIT 01 FIXTURE 1 INPUT PART B PRESENT FACE R UP MEMORY
      INPUT_PART_C_PRESENT_FACE_R_MEM : Bool;   // UNIT 01 FIXTURE 1 INPUT PART C PRESENT FACE R UP MEMORY
      INPUT_PART_D_PRESENT_FACE_R_MEM : Bool;   // UNIT 01 FIXTURE 1 INPUT PART D PRESENT FACE R UP MEMORY
      CLAMPED_WITH_PART_A : Bool;   // UNIT 01 FIXTURE 1 CLAMPED WITH PART A
      CLAMPED_WITH_PART_B : Bool;   // UNIT 01 FIXTURE 1 CLAMPED WITH PART B
      CLAMPED_WITH_PART_C : Bool;   // UNIT 01 FIXTURE 1 CLAMPED WITH PART C
      CLAMPED_WITH_PART_D : Bool;   // UNIT 01 FIXTURE 1 CLAMPED WITH PART D
      CLAMPED_WITHOUT_PART_A : Bool;   // UNIT 01 FIXTURE 1 CLAMPED WITHOUT PART A
      CLAMPED_WITHOUT_PART_B : Bool;   // UNIT 01 FIXTURE 1 CLAMPED WITHOUT PART B
      CLAMPED_WITHOUT_PART_C : Bool;   // UNIT 01 FIXTURE 1 CLAMPED WITHOUT PART C
      CLAMPED_WITHOUT_PART_D : Bool;   // UNIT 01 FIXTURE 1 CLAMPED WITHOUT PART D
      CLAMPED_WITH_PARTS : Bool;   // UNIT 01 FIXTURE 1 CLAMPED WITH PARTS
      CLAMPED_WITHOUT_PARTS : Bool;   // UNIT 01 FIXTURE 1 CLAMPED WITHOUT PARTS
      PARTIAL_CLAMPED : Bool;   // UNIT 01 FIXTURE 1 PARTIAL CLAMPED
      CLAMPED_WITH_PART_ANALOG : Bool;   // UNIT 01 FIXTURE 1 CLAMPED WITH PART ANALOG
      CLAMPED_OK : Bool;   // UNIT 01 FIXTURE 1 CLAMPED OK
      CLAMPED_DELAYED : Bool;   // UNIT 01 FIXTURE 1 CLAMPED DELAYED
      CLAMPED_WITHOUT_PART_ANALOG : Bool;   // UNIT 01 FIXTURE 1 CLAMPED WITHOUT PART ANALOG
      UNCLAMPED_ANALOG : Bool;   // UNIT 01 FIXTURE 1 UNCLAMPED
      ALL_CNC_PLC_VARIABLES_ZERO : Bool;   // UNIT 01 FIXTURE 1 ALL CNC PLC VARIABLES ZERO
      FIXTURE_NOT_CLAMPED_ALARM : Bool;   // UNIT 01 FIXTURE 1 NOT CLAMPED DURING MACHINING ALARM
      PART_A_PRESENT_DISCORDANCY : Bool;   // UNIT 01 FIXTURE 1 PART A PRESENT DISCORDANCY
      PART_B_PRESENT_DISCORDANCY : Bool;   // UNIT 01 FIXTURE 1 PART B PRESENT DISCORDANCY
      PART_C_PRESENT_DISCORDANCY : Bool;   // UNIT 01 FIXTURE 1 PART C PRESENT DISCORDANCY
      PART_D_PRESENT_DISCORDANCY : Bool;   // UNIT 01 FIXTURE 1 PART D PRESENT DISCORDANCY
      PART_A_ORIENTATED_DISCORDANCY : Bool;   // UNIT 01 FIXTURE 1 PART A ORIENTATED DISCORDANCY
      PART_B_ORIENTATED_DISCORDANCY : Bool;   // UNIT 01 FIXTURE 1 PART B ORIENTATED DISCORDANCY
      PART_C_ORIENTATED_DISCORDANCY : Bool;   // UNIT 01 FIXTURE 1 PART C ORIENTATED DISCORDANCY
      PART_D_ORIENTATED_DISCORDANCY : Bool;   // UNIT 01 FIXTURE 1 PART D ORIENTATED DISCORDANCY
      PART_TYPE_DISCORDANCY : Bool;   // UNIT 01 FIXTURE 1 PART TYPE DISCORDANCY
      ANY_PART_PRESENT : Bool;   // UNIT 01 FIXTURE 1 ANY PART PRESENT
      CLAMPED_MEMORY_DONE : Bool;   // UNIT 01 FIXTURE 1 CLAMPED MEMORY DONE
      AUX_1 : Bool;
      AUX_2 : Bool;
      AUX_3 : Bool;
      TIMER_CLAMPED_DELAY : TON_TIME;   // UNIT 01 FIXTURE 1 CLAMPED TIMER
      TIMER_PART_A_ORIENTATION { S7_SetPoint := 'True'} : TON_TIME;   // UNIT 01 FIXTURE 1 PART A ORIENTATION TIMER
      TIMER_PART_A_DISCORDANCY { S7_SetPoint := 'True'} : TON_TIME;   // UNIT 01 FIXTURE 1 PART A DISCORDANCY TIMER
      TIMER_PART_C_ORIENTATION { S7_SetPoint := 'True'} : TON_TIME;   // UNIT 01 FIXTURE 1 PART C ORIENTATION TIMER
      TIMER_PART_D_ORIENTATION { S7_SetPoint := 'True'} : TON_TIME;   // UNIT 01 FIXTURE 1 PART D ORIENTATION TIMER
      TIMER_CLAMPED_WITH_ANALOG { S7_SetPoint := 'True'} : TOF_TIME;
   END_VAR
BEGIN
   TIMER_PART_A_ORIENTATION.PT := T#750ms;
   TIMER_PART_A_DISCORDANCY.PT := T#750ms;
   TIMER_PART_C_ORIENTATION.PT := T#200ms;
   TIMER_PART_D_ORIENTATION.PT := T#200ms;
   TIMER_CLAMPED_WITH_ANALOG.PT := T#100ms;
END_DATA_BLOCK

DATA_BLOCK "DB2600_UNIT_01_FIXTURE_2"   // DB2600
{ S7_Optimized_Access := 'FALSE'; DB_Accessible_From_OPC_UA := 'FALSE' }
AUTHOR : ETXETAR
VERSION : 1.0
// stored: AutoNumber false, DBAccessibleFromOPCUA false, DBAccessibleFromWebserver true, IsOnlyStoredInLoadMemory false, IsWriteProtectedInAS false
   VAR RETAIN
      INPUT_PART_A_PRESENT : Bool;   // UNIT 01 FIXTURE 2 INPUT PART A PRESENT
      INPUT_PART_B_PRESENT : Bool;   // UNIT 01 FIXTURE 2 INPUT PART B PRESENT
      INPUT_PART_C_PRESENT : Bool;   // UNIT 01 FIXTURE 2 INPUT PART C PRESENT
      INPUT_PART_D_PRESENT : Bool;   // UNIT 01 FIXTURE 2 INPUT PART D PRESENT
      INPUT_PART_A_PRESENT_FACE_N : Bool;   // UNIT 01 FIXTURE 2 INPUT PART A PRESENT FACE N UP
      INPUT_PART_B_PRESENT_FACE_N : Bool;   // UNIT 01 FIXTURE 2 INPUT PART B PRESENT FACE N UP
      INPUT_PART_C_PRESENT_FACE_N : Bool;   // UNIT 01 FIXTURE 2 INPUT PART C PRESENT FACE N UP
      INPUT_PART_D_PRESENT_FACE_N : Bool;   // UNIT 01 FIXTURE 2 INPUT PART D PRESENT FACE N UP
      INPUT_PART_A_PRESENT_FACE_R : Bool;   // UNIT 01 FIXTURE 2 INPUT PART A PRESENT FACE R UP
      INPUT_PART_B_PRESENT_FACE_R : Bool;   // UNIT 01 FIXTURE 2 INPUT PART B PRESENT FACE R UP
      INPUT_PART_C_PRESENT_FACE_R : Bool;   // UNIT 01 FIXTURE 2 INPUT PART C PRESENT FACE R UP
      INPUT_PART_D_PRESENT_FACE_R : Bool;   // UNIT 01 FIXTURE 2 INPUT PART D PRESENT FACE R UP
      INPUT_PART_A_PRESENT_MEM : Bool;   // UNIT 01 FIXTURE 2 INPUT PART A PRESENT MEMORY
      INPUT_PART_B_PRESENT_MEM : Bool;   // UNIT 01 FIXTURE 2 INPUT PART B PRESENT MEMORY
      INPUT_PART_C_PRESENT_MEM : Bool;   // UNIT 01 FIXTURE 2 INPUT PART C PRESENT MEMORY
      INPUT_PART_D_PRESENT_MEM : Bool;   // UNIT 01 FIXTURE 2 INPUT PART D PRESENT MEMORY
      INPUT_PART_A_PRESENT_FACE_N_MEM : Bool;   // UNIT 01 FIXTURE 2 INPUT PART A PRESENT FACE N UP MEMORY
      INPUT_PART_B_PRESENT_FACE_N_MEM : Bool;   // UNIT 01 FIXTURE 2 INPUT PART B PRESENT FACE N UP MEMORY
      INPUT_PART_C_PRESENT_FACE_N_MEM : Bool;   // UNIT 01 FIXTURE 2 INPUT PART C PRESENT FACE N UP MEMORY
      INPUT_PART_D_PRESENT_FACE_N_MEM : Bool;   // UNIT 01 FIXTURE 2 INPUT PART D PRESENT FACE N UP MEMORY
      INPUT_PART_A_PRESENT_FACE_R_MEM : Bool;   // UNIT 01 FIXTURE 2 INPUT PART A PRESENT FACE R UP MEMORY
      INPUT_PART_B_PRESENT_FACE_R_MEM : Bool;   // UNIT 01 FIXTURE 2 INPUT PART B PRESENT FACE R UP MEMORY
      INPUT_PART_C_PRESENT_FACE_R_MEM : Bool;   // UNIT 01 FIXTURE 2 INPUT PART C PRESENT FACE R UP MEMORY
      INPUT_PART_D_PRESENT_FACE_R_MEM : Bool;   // UNIT 01 FIXTURE 2 INPUT PART D PRESENT FACE R UP MEMORY
      CLAMPED_WITH_PART_A : Bool;   // UNIT 01 FIXTURE 2 CLAMPED WITH PART A
      CLAMPED_WITH_PART_B : Bool;   // UNIT 01 FIXTURE 2 CLAMPED WITH PART B
      CLAMPED_WITH_PART_C : Bool;   // UNIT 01 FIXTURE 2 CLAMPED WITH PART C
      CLAMPED_WITH_PART_D : Bool;   // UNIT 01 FIXTURE 2 CLAMPED WITH PART D
      CLAMPED_WITHOUT_PART_A : Bool;   // UNIT 01 FIXTURE 2 CLAMPED WITHOUT PART A
      CLAMPED_WITHOUT_PART_B : Bool;   // UNIT 01 FIXTURE 2 CLAMPED WITHOUT PART B
      CLAMPED_WITHOUT_PART_C : Bool;   // UNIT 01 FIXTURE 2 CLAMPED WITHOUT PART C
      CLAMPED_WITHOUT_PART_D : Bool;   // UNIT 01 FIXTURE 2 CLAMPED WITHOUT PART D
      CLAMPED_WITH_PARTS : Bool;   // UNIT 01 FIXTURE 2 CLAMPED WITH PARTS
      CLAMPED_WITHOUT_PARTS : Bool;   // UNIT 01 FIXTURE 2 CLAMPED WITHOUT PARTS
      PARTIAL_CLAMPED : Bool;   // UNIT 01 FIXTURE 2 PARTIAL CLAMPED
      CLAMPED_WITH_PART_ANALOG : Bool;   // UNIT 01 FIXTURE 2 CLAMPED
      CLAMPED_OK : Bool;   // UNIT 01 FIXTURE 2 CLAMPED OK
      CLAMPED_DELAYED : Bool;   // UNIT 01 FIXTURE 2 CLAMPED DELAYED
      CLAMPED_WITHOUT_PART_ANALOG : Bool;   // UNIT 01 FIXTURE 2 PARTIAL UNCLAMPED
      UNCLAMPED_ANALOG : Bool;   // UNIT 01 FIXTURE 2 UNCLAMPED
      ALL_CNC_PLC_VARIABLES_ZERO : Bool;   // UNIT 01 FIXTURE 2 ALL CNC PLC VARIABLES ZERO
      FIXTURE_NOT_CLAMPED_ALARM : Bool;   // UNIT 01 FIXTURE 2 NOT CLAMPED DURING MACHINING ALARM
      PART_A_PRESENT_DISCORDANCY : Bool;   // UNIT 01 FIXTURE 2 PART A PRESENT DISCORDANCY
      PART_B_PRESENT_DISCORDANCY : Bool;   // UNIT 01 FIXTURE 2 PART B PRESENT DISCORDANCY
      PART_C_PRESENT_DISCORDANCY : Bool;   // UNIT 01 FIXTURE 2 PART C PRESENT DISCORDANCY
      PART_D_PRESENT_DISCORDANCY : Bool;   // UNIT 01 FIXTURE 2 PART D PRESENT DISCORDANCY
      PART_A_ORIENTATED_DISCORDANCY : Bool;   // UNIT 01 FIXTURE 2 PART A ORIENTATED DISCORDANCY
      PART_B_ORIENTATED_DISCORDANCY : Bool;   // UNIT 01 FIXTURE 2 PART B ORIENTATED DISCORDANCY
      PART_C_ORIENTATED_DISCORDANCY : Bool;   // UNIT 01 FIXTURE 2 PART C ORIENTATED DISCORDANCY
      PART_D_ORIENTATED_DISCORDANCY : Bool;   // UNIT 01 FIXTURE 2 PART D ORIENTATED DISCORDANCY
      PART_TYPE_DISCORDANCY : Bool;   // UNIT 01 FIXTURE 2 PART TYPE DISCORDANCY
      ANY_PART_PRESENT : Bool;   // UNIT 01 FIXTURE 2 ANY PART PRESENT
      CLAMPED_MEMORY_DONE : Bool;   // UNIT 01 FIXTURE 2 CLAMPED MEMORY DONE
      AUX_1 : Bool;
      AUX_2 : Bool;
      AUX_3 : Bool;
      TIMER_CLAMPED_DELAY : TON_TIME;   // UNIT 01 FIXTURE 2 CLAMPED TIMER
      TIMER_PART_A_ORIENTATION { S7_SetPoint := 'True'} : TON_TIME;   // UNIT 01 FIXTURE 2 PART A ORIENTATION TIMER
      TIMER_PART_A_DISCORDANCY { S7_SetPoint := 'True'} : TON_TIME;   // UNIT 01 FIXTURE 2 PART A DISCORDANCY TIMER
      TIMER_PART_C_ORIENTATION { S7_SetPoint := 'True'} : TON_TIME;   // UNIT 01 FIXTURE 2 PART C ORIENTATION TIMER
      TIMER_PART_D_ORIENTATION { S7_SetPoint := 'True'} : TON_TIME;   // UNIT 01 FIXTURE 2 PART D ORIENTATION TIMER
      TIMER_CLAMPED_WITH_ANALOG { S7_SetPoint := 'True'} : TOF_TIME;
   END_VAR
BEGIN
   TIMER_PART_A_ORIENTATION.PT := T#750ms;
   TIMER_PART_A_DISCORDANCY.PT := T#750ms;
   TIMER_PART_C_ORIENTATION.PT := T#200ms;
   TIMER_PART_D_ORIENTATION.PT := T#200ms;
   TIMER_CLAMPED_WITH_ANALOG.PT := T#100ms;
END_DATA_BLOCK

DATA_BLOCK "DB2700_UNIT_01_FIXTURE_3"   // DB2700
{ S7_Optimized_Access := 'FALSE'; DB_Accessible_From_OPC_UA := 'FALSE' }
AUTHOR : ETXETAR
VERSION : 1.0
// stored: AutoNumber false, DBAccessibleFromOPCUA false, DBAccessibleFromWebserver true, IsOnlyStoredInLoadMemory false, IsWriteProtectedInAS false
   VAR RETAIN
      INPUT_PART_A_PRESENT : Bool;   // UNIT 01 FIXTURE 3 INPUT PART A PRESENT
      INPUT_PART_B_PRESENT : Bool;   // UNIT 01 FIXTURE 3 INPUT PART B PRESENT
      INPUT_PART_C_PRESENT : Bool;   // UNIT 01 FIXTURE 3 INPUT PART C PRESENT
      INPUT_PART_D_PRESENT : Bool;   // UNIT 01 FIXTURE 3 INPUT PART D PRESENT
      INPUT_PART_A_PRESENT_FACE_N : Bool;   // UNIT 01 FIXTURE 3 INPUT PART A PRESENT FACE N UP
      INPUT_PART_B_PRESENT_FACE_N : Bool;   // UNIT 01 FIXTURE 3 INPUT PART B PRESENT FACE N UP
      INPUT_PART_C_PRESENT_FACE_N : Bool;   // UNIT 01 FIXTURE 3 INPUT PART C PRESENT FACE N UP
      INPUT_PART_D_PRESENT_FACE_N : Bool;   // UNIT 01 FIXTURE 3 INPUT PART D PRESENT FACE N UP
      INPUT_PART_A_PRESENT_FACE_R : Bool;   // UNIT 01 FIXTURE 3 INPUT PART A PRESENT FACE R UP
      INPUT_PART_B_PRESENT_FACE_R : Bool;   // UNIT 01 FIXTURE 3 INPUT PART B PRESENT FACE R UP
      INPUT_PART_C_PRESENT_FACE_R : Bool;   // UNIT 01 FIXTURE 3 INPUT PART C PRESENT FACE R UP
      INPUT_PART_D_PRESENT_FACE_R : Bool;   // UNIT 01 FIXTURE 3 INPUT PART D PRESENT FACE R UP
      INPUT_PART_A_PRESENT_MEM : Bool;   // UNIT 01 FIXTURE 3 INPUT PART A PRESENT MEMORY
      INPUT_PART_B_PRESENT_MEM : Bool;   // UNIT 01 FIXTURE 3 INPUT PART B PRESENT MEMORY
      INPUT_PART_C_PRESENT_MEM : Bool;   // UNIT 01 FIXTURE 3 INPUT PART C PRESENT MEMORY
      INPUT_PART_D_PRESENT_MEM : Bool;   // UNIT 01 FIXTURE 3 INPUT PART D PRESENT MEMORY
      INPUT_PART_A_PRESENT_FACE_N_MEM : Bool;   // UNIT 01 FIXTURE 3 INPUT PART A PRESENT FACE N UP MEMORY
      INPUT_PART_B_PRESENT_FACE_N_MEM : Bool;   // UNIT 01 FIXTURE 3 INPUT PART B PRESENT FACE N UP MEMORY
      INPUT_PART_C_PRESENT_FACE_N_MEM : Bool;   // UNIT 01 FIXTURE 3 INPUT PART C PRESENT FACE N UP MEMORY
      INPUT_PART_D_PRESENT_FACE_N_MEM : Bool;   // UNIT 01 FIXTURE 3 INPUT PART D PRESENT FACE N UP MEMORY
      INPUT_PART_A_PRESENT_FACE_R_MEM : Bool;   // UNIT 01 FIXTURE 3 INPUT PART A PRESENT FACE R UP MEMORY
      INPUT_PART_B_PRESENT_FACE_R_MEM : Bool;   // UNIT 01 FIXTURE 3 INPUT PART B PRESENT FACE R UP MEMORY
      INPUT_PART_C_PRESENT_FACE_R_MEM : Bool;   // UNIT 01 FIXTURE 3 INPUT PART C PRESENT FACE R UP MEMORY
      INPUT_PART_D_PRESENT_FACE_R_MEM : Bool;   // UNIT 01 FIXTURE 3 INPUT PART D PRESENT FACE R UP MEMORY
      CLAMPED_WITH_PART_A : Bool;   // UNIT 01 FIXTURE 3 CLAMPED WITH PART A
      CLAMPED_WITH_PART_B : Bool;   // UNIT 01 FIXTURE 3 CLAMPED WITH PART B
      CLAMPED_WITH_PART_C : Bool;   // UNIT 01 FIXTURE 3 CLAMPED WITH PART C
      CLAMPED_WITH_PART_D : Bool;   // UNIT 01 FIXTURE 3 CLAMPED WITH PART D
      CLAMPED_WITHOUT_PART_A : Bool;   // UNIT 01 FIXTURE 3 CLAMPED WITHOUT PART A
      CLAMPED_WITHOUT_PART_B : Bool;   // UNIT 01 FIXTURE 3 CLAMPED WITHOUT PART B
      CLAMPED_WITHOUT_PART_C : Bool;   // UNIT 01 FIXTURE 3 CLAMPED WITHOUT PART C
      CLAMPED_WITHOUT_PART_D : Bool;   // UNIT 01 FIXTURE 3 CLAMPED WITHOUT PART D
      CLAMPED_WITH_PARTS : Bool;   // UNIT 01 FIXTURE 3 CLAMPED WITH PARTS
      CLAMPED_WITHOUT_PARTS : Bool;   // UNIT 01 FIXTURE 3 CLAMPED WITHOUT PARTS
      PARTIAL_CLAMPED : Bool;   // UNIT 01 FIXTURE 3 PARTIAL CLAMPED
      CLAMPED_WITH_PART_ANALOG : Bool;   // UNIT 01 FIXTURE 3 CLAMPED
      CLAMPED_OK : Bool;   // UNIT 01 FIXTURE 3 CLAMPED OK
      CLAMPED_DELAYED : Bool;   // UNIT 01 FIXTURE 3 CLAMPED DELAYED
      CLAMPED_WITHOUT_PART_ANALOG : Bool;   // UNIT 01 FIXTURE 3 PARTIAL UNCLAMPED
      UNCLAMPED_ANALOG : Bool;   // UNIT 01 FIXTURE 3 UNCLAMPED
      ALL_CNC_PLC_VARIABLES_ZERO : Bool;   // UNIT 01 FIXTURE 3 ALL CNC PLC VARIABLES ZERO
      FIXTURE_NOT_CLAMPED_ALARM : Bool;   // UNIT 01 FIXTURE 3 NOT CLAMPED DURING MACHINING ALARM
      PART_A_PRESENT_DISCORDANCY : Bool;   // UNIT 01 FIXTURE 3 PART A PRESENT DISCORDANCY
      PART_B_PRESENT_DISCORDANCY : Bool;   // UNIT 01 FIXTURE 3 PART B PRESENT DISCORDANCY
      PART_C_PRESENT_DISCORDANCY : Bool;   // UNIT 01 FIXTURE 3 PART C PRESENT DISCORDANCY
      PART_D_PRESENT_DISCORDANCY : Bool;   // UNIT 01 FIXTURE 3 PART D PRESENT DISCORDANCY
      PART_A_ORIENTATED_DISCORDANCY : Bool;   // UNIT 01 FIXTURE 3 PART A ORIENTATED DISCORDANCY
      PART_B_ORIENTATED_DISCORDANCY : Bool;   // UNIT 01 FIXTURE 3 PART B ORIENTATED DISCORDANCY
      PART_C_ORIENTATED_DISCORDANCY : Bool;   // UNIT 01 FIXTURE 3 PART C ORIENTATED DISCORDANCY
      PART_D_ORIENTATED_DISCORDANCY : Bool;   // UNIT 01 FIXTURE 3 PART D ORIENTATED DISCORDANCY
      PART_TYPE_DISCORDANCY : Bool;   // UNIT 01 FIXTURE 3 PART TYPE DISCORDANCY
      ANY_PART_PRESENT : Bool;   // UNIT 01 FIXTURE 3 ANY PART PRESENT
      CLAMPED_MEMORY_DONE : Bool;   // UNIT 01 FIXTURE 3 CLAMPED MEMORY DONE
      AUX_1 : Bool;
      AUX_2 : Bool;
      AUX_3 : Bool;
      TIMER_CLAMPED_DELAY : TON_TIME;   // UNIT 01 FIXTURE 3 CLAMPED TIMER
      TIMER_PART_A_ORIENTATION { S7_SetPoint := 'True'} : TON_TIME;   // UNIT 01 FIXTURE 3 PART A ORIENTATION TIMER
      TIMER_PART_A_DISCORDANCY { S7_SetPoint := 'True'} : TON_TIME;   // UNIT 01 FIXTURE 3 PART A DISCORDANCY TIMER
      TIMER_PART_C_ORIENTATION { S7_SetPoint := 'True'} : TON_TIME;   // UNIT 01 FIXTURE 3 PART C ORIENTATION TIMER
      TIMER_PART_D_ORIENTATION { S7_SetPoint := 'True'} : TON_TIME;   // UNIT 01 FIXTURE 3 PART D ORIENTATION TIMER
      TIMER_CLAMPED_WITH_ANALOG { S7_SetPoint := 'True'} : TOF_TIME;
   END_VAR
BEGIN
   TIMER_PART_A_ORIENTATION.PT := T#750ms;
   TIMER_PART_A_DISCORDANCY.PT := T#750ms;
   TIMER_PART_C_ORIENTATION.PT := T#200ms;
   TIMER_PART_D_ORIENTATION.PT := T#200ms;
   TIMER_CLAMPED_WITH_ANALOG.PT := T#100ms;
END_DATA_BLOCK

DATA_BLOCK "DB2800_UNIT_01_FIXTURE_4"   // DB2800
{ S7_Optimized_Access := 'FALSE'; DB_Accessible_From_OPC_UA := 'FALSE' }
AUTHOR : ETXETAR
VERSION : 1.0
// stored: AutoNumber false, DBAccessibleFromOPCUA false, DBAccessibleFromWebserver true, IsOnlyStoredInLoadMemory false, IsWriteProtectedInAS false
   VAR RETAIN
      INPUT_PART_A_PRESENT : Bool;   // UNIT 01 FIXTURE 4 INPUT PART A PRESENT
      INPUT_PART_B_PRESENT : Bool;   // UNIT 01 FIXTURE 4 INPUT PART B PRESENT
      INPUT_PART_C_PRESENT : Bool;   // UNIT 01 FIXTURE 4 INPUT PART C PRESENT
      INPUT_PART_D_PRESENT : Bool;   // UNIT 01 FIXTURE 4 INPUT PART D PRESENT
      INPUT_PART_A_PRESENT_FACE_N : Bool;   // UNIT 01 FIXTURE 4 INPUT PART A PRESENT FACE N UP
      INPUT_PART_B_PRESENT_FACE_N : Bool;   // UNIT 01 FIXTURE 4 INPUT PART B PRESENT FACE N UP
      INPUT_PART_C_PRESENT_FACE_N : Bool;   // UNIT 01 FIXTURE 4 INPUT PART C PRESENT FACE N UP
      INPUT_PART_D_PRESENT_FACE_N : Bool;   // UNIT 01 FIXTURE 4 INPUT PART D PRESENT FACE N UP
      INPUT_PART_A_PRESENT_FACE_R : Bool;   // UNIT 01 FIXTURE 4 INPUT PART A PRESENT FACE R UP
      INPUT_PART_B_PRESENT_FACE_R : Bool;   // UNIT 01 FIXTURE 4 INPUT PART B PRESENT FACE R UP
      INPUT_PART_C_PRESENT_FACE_R : Bool;   // UNIT 01 FIXTURE 4 INPUT PART C PRESENT FACE R UP
      INPUT_PART_D_PRESENT_FACE_R : Bool;   // UNIT 01 FIXTURE 4 INPUT PART D PRESENT FACE R UP
      INPUT_PART_A_PRESENT_MEM : Bool;   // UNIT 01 FIXTURE 4 INPUT PART A PRESENT MEMORY
      INPUT_PART_B_PRESENT_MEM : Bool;   // UNIT 01 FIXTURE 4 INPUT PART B PRESENT MEMORY
      INPUT_PART_C_PRESENT_MEM : Bool;   // UNIT 01 FIXTURE 4 INPUT PART C PRESENT MEMORY
      INPUT_PART_D_PRESENT_MEM : Bool;   // UNIT 01 FIXTURE 4 INPUT PART D PRESENT MEMORY
      INPUT_PART_A_PRESENT_FACE_N_MEM : Bool;   // UNIT 01 FIXTURE 4 INPUT PART A PRESENT FACE N UP MEMORY
      INPUT_PART_B_PRESENT_FACE_N_MEM : Bool;   // UNIT 01 FIXTURE 4 INPUT PART B PRESENT FACE N UP MEMORY
      INPUT_PART_C_PRESENT_FACE_N_MEM : Bool;   // UNIT 01 FIXTURE 4 INPUT PART C PRESENT FACE N UP MEMORY
      INPUT_PART_D_PRESENT_FACE_N_MEM : Bool;   // UNIT 01 FIXTURE 4 INPUT PART D PRESENT FACE N UP MEMORY
      INPUT_PART_A_PRESENT_FACE_R_MEM : Bool;   // UNIT 01 FIXTURE 4 INPUT PART A PRESENT FACE R UP MEMORY
      INPUT_PART_B_PRESENT_FACE_R_MEM : Bool;   // UNIT 01 FIXTURE 4 INPUT PART B PRESENT FACE R UP MEMORY
      INPUT_PART_C_PRESENT_FACE_R_MEM : Bool;   // UNIT 01 FIXTURE 4 INPUT PART C PRESENT FACE R UP MEMORY
      INPUT_PART_D_PRESENT_FACE_R_MEM : Bool;   // UNIT 01 FIXTURE 4 INPUT PART D PRESENT FACE R UP MEMORY
      CLAMPED_WITH_PART_A : Bool;   // UNIT 01 FIXTURE 4 CLAMPED WITH PART A
      CLAMPED_WITH_PART_B : Bool;   // UNIT 01 FIXTURE 4 CLAMPED WITH PART B
      CLAMPED_WITH_PART_C : Bool;   // UNIT 01 FIXTURE 4 CLAMPED WITH PART C
      CLAMPED_WITH_PART_D : Bool;   // UNIT 01 FIXTURE 4 CLAMPED WITH PART D
      CLAMPED_WITHOUT_PART_A : Bool;   // UNIT 01 FIXTURE 4 CLAMPED WITHOUT PART A
      CLAMPED_WITHOUT_PART_B : Bool;   // UNIT 01 FIXTURE 4 CLAMPED WITHOUT PART B
      CLAMPED_WITHOUT_PART_C : Bool;   // UNIT 01 FIXTURE 4 CLAMPED WITHOUT PART C
      CLAMPED_WITHOUT_PART_D : Bool;   // UNIT 01 FIXTURE 4 CLAMPED WITHOUT PART D
      CLAMPED_WITH_PARTS : Bool;   // UNIT 01 FIXTURE 4 CLAMPED WITH PARTS
      CLAMPED_WITHOUT_PARTS : Bool;   // UNIT 01 FIXTURE 4 CLAMPED WITHOUT PARTS
      PARTIAL_CLAMPED : Bool;   // UNIT 01 FIXTURE 4 PARTIAL CLAMPED
      CLAMPED_WITH_PART_ANALOG : Bool;   // UNIT 01 FIXTURE 4 CLAMPED
      CLAMPED_OK : Bool;   // UNIT 01 FIXTURE 4 CLAMPED OK
      CLAMPED_DELAYED : Bool;   // UNIT 01 FIXTURE 4 CLAMPED DELAYED
      CLAMPED_WITHOUT_PART_ANALOG : Bool;   // UNIT 01 FIXTURE 4 PARTIAL UNCLAMPED
      UNCLAMPED_ANALOG : Bool;   // UNIT 01 FIXTURE 4 UNCLAMPED
      ALL_CNC_PLC_VARIABLES_ZERO : Bool;   // UNIT 01 FIXTURE 4 ALL CNC PLC VARIABLES ZERO
      FIXTURE_NOT_CLAMPED_ALARM : Bool;   // UNIT 01 FIXTURE 4 NOT CLAMPED DURING MACHINING ALARM
      PART_A_PRESENT_DISCORDANCY : Bool;   // UNIT 01 FIXTURE 4 PART A PRESENT DISCORDANCY
      PART_B_PRESENT_DISCORDANCY : Bool;   // UNIT 01 FIXTURE 4 PART B PRESENT DISCORDANCY
      PART_C_PRESENT_DISCORDANCY : Bool;   // UNIT 01 FIXTURE 4 PART C PRESENT DISCORDANCY
      PART_D_PRESENT_DISCORDANCY : Bool;   // UNIT 01 FIXTURE 4 PART D PRESENT DISCORDANCY
      PART_A_ORIENTATED_DISCORDANCY : Bool;   // UNIT 01 FIXTURE 4 PART A ORIENTATED DISCORDANCY
      PART_B_ORIENTATED_DISCORDANCY : Bool;   // UNIT 01 FIXTURE 4 PART B ORIENTATED DISCORDANCY
      PART_C_ORIENTATED_DISCORDANCY : Bool;   // UNIT 01 FIXTURE 4 PART C ORIENTATED DISCORDANCY
      PART_D_ORIENTATED_DISCORDANCY : Bool;   // UNIT 01 FIXTURE 4 PART D ORIENTATED DISCORDANCY
      PART_TYPE_DISCORDANCY : Bool;   // UNIT 01 FIXTURE 4 PART TYPE DISCORDANCY
      ANY_PART_PRESENT : Bool;   // UNIT 01 FIXTURE 4 ANY PART PRESENT
      CLAMPED_MEMORY_DONE : Bool;   // UNIT 01 FIXTURE 4 CLAMPED MEMORY DONE
      AUX_1 : Bool;
      AUX_2 : Bool;
      AUX_3 : Bool;
      TIMER_CLAMPED_DELAY : TON_TIME;   // UNIT 01 FIXTURE 4 CLAMPED TIMER
      TIMER_PART_A_ORIENTATION { S7_SetPoint := 'True'} : TON_TIME;   // UNIT 01 FIXTURE 4 PART A ORIENTATION TIMER
      TIMER_PART_A_DISCORDANCY { S7_SetPoint := 'True'} : TON_TIME;   // UNIT 01 FIXTURE 4 PART A DISCORDANCY TIMER
      TIMER_PART_C_ORIENTATION { S7_SetPoint := 'True'} : TON_TIME;   // UNIT 01 FIXTURE 4 PART C ORIENTATION TIMER
      TIMER_PART_D_ORIENTATION { S7_SetPoint := 'True'} : TON_TIME;   // UNIT 01 FIXTURE 4 PART D ORIENTATION TIMER
      TIMER_CLAMPED_WITH_ANALOG { S7_SetPoint := 'True'} : TOF_TIME;
   END_VAR
BEGIN
   TIMER_PART_A_ORIENTATION.PT := T#750ms;
   TIMER_PART_A_DISCORDANCY.PT := T#750ms;
   TIMER_PART_C_ORIENTATION.PT := T#200ms;
   TIMER_PART_D_ORIENTATION.PT := T#200ms;
   TIMER_CLAMPED_WITH_ANALOG.PT := T#100ms;
END_DATA_BLOCK

DATA_BLOCK "DB3500_UNIT_02_FIXTURE_1"   // DB3500
{ S7_Optimized_Access := 'FALSE'; DB_Accessible_From_OPC_UA := 'FALSE' }
AUTHOR : ETXETAR
VERSION : 1.0
// stored: AutoNumber false, DBAccessibleFromOPCUA false, DBAccessibleFromWebserver true, IsOnlyStoredInLoadMemory false, IsWriteProtectedInAS false
   VAR RETAIN
      INPUT_PART_A_PRESENT : Bool;   // UNIT 02 FIXTURE 1 INPUT PART A PRESENT
      INPUT_PART_B_PRESENT : Bool;   // UNIT 02 FIXTURE 1 INPUT PART B PRESENT
      INPUT_PART_C_PRESENT : Bool;   // UNIT 02 FIXTURE 1 INPUT PART C PRESENT
      INPUT_PART_D_PRESENT : Bool;   // UNIT 02 FIXTURE 1 INPUT PART D PRESENT
      INPUT_PART_A_PRESENT_FACE_N : Bool;   // UNIT 02 FIXTURE 1 INPUT PART A PRESENT FACE N UP
      INPUT_PART_B_PRESENT_FACE_N : Bool;   // UNIT 02 FIXTURE 1 INPUT PART B PRESENT FACE N UP
      INPUT_PART_C_PRESENT_FACE_N : Bool;   // UNIT 02 FIXTURE 1 INPUT PART C PRESENT FACE N UP
      INPUT_PART_D_PRESENT_FACE_N : Bool;   // UNIT 02 FIXTURE 1 INPUT PART D PRESENT FACE N UP
      INPUT_PART_A_PRESENT_FACE_R : Bool;   // UNIT 02 FIXTURE 1 INPUT PART A PRESENT FACE R UP
      INPUT_PART_B_PRESENT_FACE_R : Bool;   // UNIT 02 FIXTURE 1 INPUT PART B PRESENT FACE R UP
      INPUT_PART_C_PRESENT_FACE_R : Bool;   // UNIT 02 FIXTURE 1 INPUT PART C PRESENT FACE R UP
      INPUT_PART_D_PRESENT_FACE_R : Bool;   // UNIT 02 FIXTURE 1 INPUT PART D PRESENT FACE R UP
      INPUT_PART_A_PRESENT_MEM : Bool;   // UNIT 02 FIXTURE 1 INPUT PART A PRESENT MEMORY
      INPUT_PART_B_PRESENT_MEM : Bool;   // UNIT 02 FIXTURE 1 INPUT PART B PRESENT MEMORY
      INPUT_PART_C_PRESENT_MEM : Bool;   // UNIT 02 FIXTURE 1 INPUT PART C PRESENT MEMORY
      INPUT_PART_D_PRESENT_MEM : Bool;   // UNIT 02 FIXTURE 1 INPUT PART D PRESENT MEMORY
      INPUT_PART_A_PRESENT_FACE_N_MEM : Bool;   // UNIT 02 FIXTURE 1 INPUT PART A PRESENT FACE A UP MEMORY
      INPUT_PART_B_PRESENT_FACE_N_MEM : Bool;   // UNIT 02 FIXTURE 1 INPUT PART B PRESENT FACE N UP MEMORY
      INPUT_PART_C_PRESENT_FACE_N_MEM : Bool;   // UNIT 02 FIXTURE 1 INPUT PART C PRESENT FACE N UP MEMORY
      INPUT_PART_D_PRESENT_FACE_N_MEM : Bool;   // UNIT 02 FIXTURE 1 INPUT PART D PRESENT FACE N UP MEMORY
      INPUT_PART_A_PRESENT_FACE_R_MEM : Bool;   // UNIT 02 FIXTURE 1 INPUT PART A PRESENT FACE R UP MEMORY
      INPUT_PART_B_PRESENT_FACE_R_MEM : Bool;   // UNIT 02 FIXTURE 1 INPUT PART B PRESENT FACE R UP MEMORY
      INPUT_PART_C_PRESENT_FACE_R_MEM : Bool;   // UNIT 02 FIXTURE 1 INPUT PART C PRESENT FACE R UP MEMORY
      INPUT_PART_D_PRESENT_FACE_R_MEM : Bool;   // UNIT 02 FIXTURE 1 INPUT PART D PRESENT FACE R UP MEMORY
      CLAMPED_WITH_PART_A : Bool;   // UNIT 02 FIXTURE 1 CLAMPED WITH PART A
      CLAMPED_WITH_PART_B : Bool;   // UNIT 02 FIXTURE 1 CLAMPED WITH PART B
      CLAMPED_WITH_PART_C : Bool;   // UNIT 02 FIXTURE 1 CLAMPED WITH PART C
      CLAMPED_WITH_PART_D : Bool;   // UNIT 02 FIXTURE 1 CLAMPED WITH PART D
      CLAMPED_WITHOUT_PART_A : Bool;   // UNIT 02 FIXTURE 1 CLAMPED WITHOUT PART A
      CLAMPED_WITHOUT_PART_B : Bool;   // UNIT 02 FIXTURE 1 CLAMPED WITHOUT PART B
      CLAMPED_WITHOUT_PART_C : Bool;   // UNIT 02 FIXTURE 1 CLAMPED WITHOUT PART C
      CLAMPED_WITHOUT_PART_D : Bool;   // UNIT 02 FIXTURE 1 CLAMPED WITHOUT PART D
      CLAMPED_WITH_PARTS : Bool;   // UNIT 02 FIXTURE 1 CLAMPED WITH PARTS
      CLAMPED_WITHOUT_PARTS : Bool;   // UNIT 02 FIXTURE 1 CLAMPED WITHOUT PARTS
      PARTIAL_CLAMPED : Bool;   // UNIT 02 FIXTURE 1 PARTIAL CLAMPED
      CLAMPED_WITH_PART_ANALOG : Bool;   // UNIT 02 FIXTURE 1 CLAMPED
      CLAMPED_OK : Bool;   // UNIT 02 FIXTURE 1 CLAMPED OK
      CLAMPED_DELAYED : Bool;   // UNIT 02 FIXTURE 1 CLAMPED DELAYED
      CLAMPED_WITHOUT_PART_ANALOG : Bool;   // UNIT 02 FIXTURE 1 PARTIAL UNCLAMPED
      UNCLAMPED_ANALOG : Bool;   // UNIT 02 FIXTURE 1 UNCLAMPED
      ALL_CNC_PLC_VARIABLES_ZERO : Bool;   // UNIT 02 FIXTURE 1 ALL CNC PLC VARIABLES ZERO
      FIXTURE_NOT_CLAMPED_ALARM : Bool;   // UNIT 02 FIXTURE 1 NOT CLAMPED DURING MACHINING ALARM
      PART_A_PRESENT_DISCORDANCY : Bool;   // UNIT 02 FIXTURE 1 PART A PRESENT DISCORDANCY
      PART_B_PRESENT_DISCORDANCY : Bool;   // UNIT 02 FIXTURE 1 PART B PRESENT DISCORDANCY
      PART_C_PRESENT_DISCORDANCY : Bool;   // UNIT 02 FIXTURE 1 PART C PRESENT DISCORDANCY
      PART_D_PRESENT_DISCORDANCY : Bool;   // UNIT 02 FIXTURE 1 PART D PRESENT DISCORDANCY
      PART_A_ORIENTATED_DISCORDANCY : Bool;   // UNIT 02 FIXTURE 1 PART A ORIENTATED DISCORDANCY
      PART_B_ORIENTATED_DISCORDANCY : Bool;   // UNIT 02 FIXTURE 1 PART B ORIENTATED DISCORDANCY
      PART_C_ORIENTATED_DISCORDANCY : Bool;   // UNIT 02 FIXTURE 1 PART C ORIENTATED DISCORDANCY
      PART_D_ORIENTATED_DISCORDANCY : Bool;   // UNIT 02 FIXTURE 1 PART D ORIENTATED DISCORDANCY
      PART_TYPE_DISCORDANCY : Bool;   // UNIT 02 FIXTURE 1 PART TYPE DISCORDANCY
      ANY_PART_PRESENT : Bool;   // UNIT 02 FIXTURE 1 ANY PART PRESENT
      CLAMPED_MEMORY_DONE : Bool;   // UNIT 02 FIXTURE 1 CLAMPED MEMORY DONE
      AUX_1 : Bool;
      AUX_2 : Bool;
      AUX_3 : Bool;
      TIMER_CLAMPED_DELAY : TON_TIME;   // UNIT 02 FIXTURE 1 CLAMPED TIMER
      TIMER_PART_A_ORIENTATION { S7_SetPoint := 'True'} : TON_TIME;   // UNIT 02 FIXTURE 1 PART A ORIENTATION TIMER
      TIMER_PART_A_DISCORDANCY { S7_SetPoint := 'True'} : TON_TIME;   // UNIT 02 FIXTURE 1 PART A DISCORDANCY TIMER
      TIMER_PART_C_ORIENTATION { S7_SetPoint := 'True'} : TON_TIME;   // UNIT 02 FIXTURE 1 PART C ORIENTATION TIMER
      TIMER_PART_D_ORIENTATION { S7_SetPoint := 'True'} : TON_TIME;   // UNIT 02 FIXTURE 1 PART D ORIENTATION TIMER
      TIMER_CLAMPED_WITH_ANALOG { S7_SetPoint := 'True'} : TOF_TIME;
   END_VAR
BEGIN
   TIMER_PART_A_ORIENTATION.PT := T#200ms;
   TIMER_PART_A_DISCORDANCY.PT := T#200ms;
   TIMER_PART_C_ORIENTATION.PT := T#200ms;
   TIMER_PART_D_ORIENTATION.PT := T#200ms;
   TIMER_CLAMPED_WITH_ANALOG.PT := T#100ms;
END_DATA_BLOCK

DATA_BLOCK "DB3600_UNIT_02_FIXTURE_2"   // DB3600
{ S7_Optimized_Access := 'FALSE'; DB_Accessible_From_OPC_UA := 'FALSE' }
AUTHOR : ETXETAR
VERSION : 1.0
// stored: AutoNumber false, DBAccessibleFromOPCUA false, DBAccessibleFromWebserver true, IsOnlyStoredInLoadMemory false, IsWriteProtectedInAS false
   VAR RETAIN
      INPUT_PART_A_PRESENT : Bool;   // UNIT 02 FIXTURE 2 INPUT PART A PRESENT
      INPUT_PART_B_PRESENT : Bool;   // UNIT 02 FIXTURE 2 INPUT PART B PRESENT
      INPUT_PART_C_PRESENT : Bool;   // UNIT 02 FIXTURE 2 INPUT PART C PRESENT
      INPUT_PART_D_PRESENT : Bool;   // UNIT 02 FIXTURE 2 INPUT PART D PRESENT
      INPUT_PART_A_PRESENT_FACE_N : Bool;   // UNIT 02 FIXTURE 2 INPUT PART A PRESENT FACE N UP
      INPUT_PART_B_PRESENT_FACE_N : Bool;   // UNIT 02 FIXTURE 2 INPUT PART B PRESENT FACE N UP
      INPUT_PART_C_PRESENT_FACE_N : Bool;   // UNIT 02 FIXTURE 2 INPUT PART C PRESENT FACE N UP
      INPUT_PART_D_PRESENT_FACE_N : Bool;   // UNIT 02 FIXTURE 2 INPUT PART D PRESENT FACE N UP
      INPUT_PART_A_PRESENT_FACE_R : Bool;   // UNIT 02 FIXTURE 2 INPUT PART A PRESENT FACE R UP
      INPUT_PART_B_PRESENT_FACE_R : Bool;   // UNIT 02 FIXTURE 2 INPUT PART B PRESENT FACE R UP
      INPUT_PART_C_PRESENT_FACE_R : Bool;   // UNIT 02 FIXTURE 2 INPUT PART C PRESENT FACE R UP
      INPUT_PART_D_PRESENT_FACE_R : Bool;   // UNIT 02 FIXTURE 2 INPUT PART D PRESENT FACE R UP
      INPUT_PART_A_PRESENT_MEM : Bool;   // UNIT 02 FIXTURE 2 INPUT PART A PRESENT MEMORY
      INPUT_PART_B_PRESENT_MEM : Bool;   // UNIT 02 FIXTURE 2 INPUT PART B PRESENT MEMORY
      INPUT_PART_C_PRESENT_MEM : Bool;   // UNIT 02 FIXTURE 2 INPUT PART C PRESENT MEMORY
      INPUT_PART_D_PRESENT_MEM : Bool;   // UNIT 02 FIXTURE 2 INPUT PART D PRESENT MEMORY
      INPUT_PART_A_PRESENT_FACE_N_MEM : Bool;   // UNIT 02 FIXTURE 2 INPUT PART A PRESENT FACE N UP MEMORY
      INPUT_PART_B_PRESENT_FACE_N_MEM : Bool;   // UNIT 02 FIXTURE 2 INPUT PART B PRESENT FACE N UP MEMORY
      INPUT_PART_C_PRESENT_FACE_N_MEM : Bool;   // UNIT 02 FIXTURE 2 INPUT PART C PRESENT FACE N UP MEMORY
      INPUT_PART_D_PRESENT_FACE_N_MEM : Bool;   // UNIT 02 FIXTURE 2 INPUT PART D PRESENT FACE N UP MEMORY
      INPUT_PART_A_PRESENT_FACE_R_MEM : Bool;   // UNIT 02 FIXTURE 2 INPUT PART A PRESENT FACE R UP MEMORY
      INPUT_PART_B_PRESENT_FACE_R_MEM : Bool;   // UNIT 02 FIXTURE 2 INPUT PART B PRESENT FACE R UP MEMORY
      INPUT_PART_C_PRESENT_FACE_R_MEM : Bool;   // UNIT 02 FIXTURE 2 INPUT PART C PRESENT FACE R UP MEMORY
      INPUT_PART_D_PRESENT_FACE_R_MEM : Bool;   // UNIT 02 FIXTURE 2 INPUT PART D PRESENT FACE R UP MEMORY
      CLAMPED_WITH_PART_A : Bool;   // UNIT 02 FIXTURE 2 CLAMPED WITH PART A
      CLAMPED_WITH_PART_B : Bool;   // UNIT 02 FIXTURE 2 CLAMPED WITH PART B
      CLAMPED_WITH_PART_C : Bool;   // UNIT 02 FIXTURE 2 CLAMPED WITH PART C
      CLAMPED_WITH_PART_D : Bool;   // UNIT 02 FIXTURE 2 CLAMPED WITH PART D
      CLAMPED_WITHOUT_PART_A : Bool;   // UNIT 02 FIXTURE 2 CLAMPED WITHOUT PART A
      CLAMPED_WITHOUT_PART_B : Bool;   // UNIT 02 FIXTURE 2 CLAMPED WITHOUT PART B
      CLAMPED_WITHOUT_PART_C : Bool;   // UNIT 02 FIXTURE 2 CLAMPED WITHOUT PART C
      CLAMPED_WITHOUT_PART_D : Bool;   // UNIT 02 FIXTURE 2 CLAMPED WITHOUT PART D
      CLAMPED_WITH_PARTS : Bool;   // UNIT 02 FIXTURE 2 CLAMPED WITH PARTS
      CLAMPED_WITHOUT_PARTS : Bool;   // UNIT 02 FIXTURE 2 CLAMPED WITHOUT PARTS
      PARTIAL_CLAMPED : Bool;   // UNIT 02 FIXTURE 2 PARTIAL CLAMPED
      CLAMPED_WITH_PART_ANALOG : Bool;   // UNIT 02 FIXTURE 2 CLAMPED
      CLAMPED_OK : Bool;   // UNIT 02 FIXTURE 2 CLAMPED OK
      CLAMPED_DELAYED : Bool;   // UNIT 02 FIXTURE 2 CLAMPED DELAYED
      CLAMPED_WITHOUT_PART_ANALOG : Bool;   // UNIT 02 FIXTURE 2 PARTIAL UNCLAMPED
      UNCLAMPED_ANALOG : Bool;   // UNIT 02 FIXTURE 2 UNCLAMPED
      ALL_CNC_PLC_VARIABLES_ZERO : Bool;   // UNIT 02 FIXTURE 2 ALL CNC PLC VARIABLES ZERO
      FIXTURE_NOT_CLAMPED_ALARM : Bool;   // UNIT 02 FIXTURE 2 NOT CLAMPED DURING MACHINING ALARM
      PART_A_PRESENT_DISCORDANCY : Bool;   // UNIT 02 FIXTURE 2 PART A PRESENT DISCORDANCY
      PART_B_PRESENT_DISCORDANCY : Bool;   // UNIT 02 FIXTURE 2 PART B PRESENT DISCORDANCY
      PART_C_PRESENT_DISCORDANCY : Bool;   // UNIT 02 FIXTURE 2 PART C PRESENT DISCORDANCY
      PART_D_PRESENT_DISCORDANCY : Bool;   // UNIT 02 FIXTURE 2 PART D PRESENT DISCORDANCY
      PART_A_ORIENTATED_DISCORDANCY : Bool;   // UNIT 02 FIXTURE 2 PART A ORIENTATED DISCORDANCY
      PART_B_ORIENTATED_DISCORDANCY : Bool;   // UNIT 02 FIXTURE 2 PART B ORIENTATED DISCORDANCY
      PART_C_ORIENTATED_DISCORDANCY : Bool;   // UNIT 02 FIXTURE 2 PART C ORIENTATED DISCORDANCY
      PART_D_ORIENTATED_DISCORDANCY : Bool;   // UNIT 02 FIXTURE 2 PART D ORIENTATED DISCORDANCY
      PART_TYPE_DISCORDANCY : Bool;   // UNIT 02 FIXTURE 2 PART TYPE DISCORDANCY
      ANY_PART_PRESENT : Bool;   // UNIT 02 FIXTURE 2 ANY PART PRESENT
      CLAMPED_MEMORY_DONE : Bool;   // UNIT 02 FIXTURE 2 CLAMPED MEMORY DONE
      AUX_1 : Bool;
      AUX_2 : Bool;
      AUX_3 : Bool;
      TIMER_CLAMPED_DELAY : TON_TIME;   // UNIT 02 FIXTURE 2 CLAMPED TIMER
      TIMER_PART_A_ORIENTATION { S7_SetPoint := 'True'} : TON_TIME;   // UNIT 02 FIXTURE 2 PART A ORIENTATION TIMER
      TIMER_PART_A_DISCORDANCY { S7_SetPoint := 'True'} : TON_TIME;   // UNIT 02 FIXTURE 2 PART A DISCORDANCY TIMER
      TIMER_PART_C_ORIENTATION { S7_SetPoint := 'True'} : TON_TIME;   // UNIT 02 FIXTURE 2 PART C ORIENTATION TIMER
      TIMER_PART_D_ORIENTATION { S7_SetPoint := 'True'} : TON_TIME;   // UNIT 02 FIXTURE 2 PART D ORIENTATION TIMER
      TIMER_CLAMPED_WITH_ANALOG { S7_SetPoint := 'True'} : TOF_TIME;
   END_VAR
BEGIN
   TIMER_PART_A_ORIENTATION.PT := T#200ms;
   TIMER_PART_A_DISCORDANCY.PT := T#200ms;
   TIMER_PART_C_ORIENTATION.PT := T#200ms;
   TIMER_PART_D_ORIENTATION.PT := T#200ms;
   TIMER_CLAMPED_WITH_ANALOG.PT := T#100ms;
END_DATA_BLOCK

DATA_BLOCK "DB3700_UNIT_02_FIXTURE_3"   // DB3700
{ S7_Optimized_Access := 'FALSE'; DB_Accessible_From_OPC_UA := 'FALSE' }
AUTHOR : ETXETAR
VERSION : 1.0
// stored: AutoNumber false, DBAccessibleFromOPCUA false, DBAccessibleFromWebserver true, IsOnlyStoredInLoadMemory false, IsWriteProtectedInAS false
   VAR RETAIN
      INPUT_PART_A_PRESENT : Bool;   // UNIT 02 FIXTURE 3 INPUT PART A PRESENT
      INPUT_PART_B_PRESENT : Bool;   // UNIT 02 FIXTURE 3 INPUT PART B PRESENT
      INPUT_PART_C_PRESENT : Bool;   // UNIT 02 FIXTURE 3 INPUT PART C PRESENT
      INPUT_PART_D_PRESENT : Bool;   // UNIT 02 FIXTURE 3 INPUT PART D PRESENT
      INPUT_PART_A_PRESENT_FACE_N : Bool;   // UNIT 02 FIXTURE 3 INPUT PART A PRESENT FACE N UP
      INPUT_PART_B_PRESENT_FACE_N : Bool;   // UNIT 02 FIXTURE 3 INPUT PART B PRESENT FACE N UP
      INPUT_PART_C_PRESENT_FACE_N : Bool;   // UNIT 02 FIXTURE 3 INPUT PART C PRESENT FACE N UP
      INPUT_PART_D_PRESENT_FACE_N : Bool;   // UNIT 02 FIXTURE 3 INPUT PART D PRESENT FACE N UP
      INPUT_PART_A_PRESENT_FACE_R : Bool;   // UNIT 02 FIXTURE 3 INPUT PART A PRESENT FACE R UP
      INPUT_PART_B_PRESENT_FACE_R : Bool;   // UNIT 02 FIXTURE 3 INPUT PART B PRESENT FACE R UP
      INPUT_PART_C_PRESENT_FACE_R : Bool;   // UNIT 02 FIXTURE 3 INPUT PART C PRESENT FACE R UP
      INPUT_PART_D_PRESENT_FACE_R : Bool;   // UNIT 02 FIXTURE 3 INPUT PART D PRESENT FACE R UP
      INPUT_PART_A_PRESENT_MEM : Bool;   // UNIT 02 FIXTURE 3 INPUT PART A PRESENT MEMORY
      INPUT_PART_B_PRESENT_MEM : Bool;   // UNIT 02 FIXTURE 3 INPUT PART B PRESENT MEMORY
      INPUT_PART_C_PRESENT_MEM : Bool;   // UNIT 02 FIXTURE 3 INPUT PART C PRESENT MEMORY
      INPUT_PART_D_PRESENT_MEM : Bool;   // UNIT 02 FIXTURE 3 INPUT PART D PRESENT MEMORY
      INPUT_PART_A_PRESENT_FACE_N_MEM : Bool;   // UNIT 02 FIXTURE 3 INPUT PART A PRESENT FACE N UP MEMORY
      INPUT_PART_B_PRESENT_FACE_N_MEM : Bool;   // UNIT 02 FIXTURE 3 INPUT PART B PRESENT FACE N UP MEMORY
      INPUT_PART_C_PRESENT_FACE_N_MEM : Bool;   // UNIT 02 FIXTURE 3 INPUT PART C PRESENT FACE N UP MEMORY
      INPUT_PART_D_PRESENT_FACE_N_MEM : Bool;   // UNIT 02 FIXTURE 3 INPUT PART D PRESENT FACE N UP MEMORY
      INPUT_PART_A_PRESENT_FACE_R_MEM : Bool;   // UNIT 02 FIXTURE 3 INPUT PART A PRESENT FACE R UP MEMORY
      INPUT_PART_B_PRESENT_FACE_R_MEM : Bool;   // UNIT 02 FIXTURE 3 INPUT PART B PRESENT FACE R UP MEMORY
      INPUT_PART_C_PRESENT_FACE_R_MEM : Bool;   // UNIT 02 FIXTURE 3 INPUT PART C PRESENT FACE R UP MEMORY
      INPUT_PART_D_PRESENT_FACE_R_MEM : Bool;   // UNIT 02 FIXTURE 3 INPUT PART D PRESENT FACE R UP MEMORY
      CLAMPED_WITH_PART_A : Bool;   // UNIT 02 FIXTURE 3 CLAMPED WITH PART A
      CLAMPED_WITH_PART_B : Bool;   // UNIT 02 FIXTURE 3 CLAMPED WITH PART B
      CLAMPED_WITH_PART_C : Bool;   // UNIT 02 FIXTURE 3 CLAMPED WITH PART C
      CLAMPED_WITH_PART_D : Bool;   // UNIT 02 FIXTURE 3 CLAMPED WITH PART D
      CLAMPED_WITHOUT_PART_A : Bool;   // UNIT 02 FIXTURE 3 CLAMPED WITHOUT PART A
      CLAMPED_WITHOUT_PART_B : Bool;   // UNIT 02 FIXTURE 3 CLAMPED WITHOUT PART B
      CLAMPED_WITHOUT_PART_C : Bool;   // UNIT 02 FIXTURE 3 CLAMPED WITHOUT PART C
      CLAMPED_WITHOUT_PART_D : Bool;   // UNIT 02 FIXTURE 3 CLAMPED WITHOUT PART D
      CLAMPED_WITH_PARTS : Bool;   // UNIT 02 FIXTURE 3 CLAMPED WITH PARTS
      CLAMPED_WITHOUT_PARTS : Bool;   // UNIT 02 FIXTURE 3 CLAMPED WITHOUT PARTS
      PARTIAL_CLAMPED : Bool;   // UNIT 02 FIXTURE 3 PARTIAL CLAMPED
      CLAMPED_WITH_PART_ANALOG : Bool;   // UNIT 02 FIXTURE 3 CLAMPED
      CLAMPED_OK : Bool;   // UNIT 02 FIXTURE 3 CLAMPED OK
      CLAMPED_DELAYED : Bool;   // UNIT 02 FIXTURE 3 CLAMPED DELAYED
      CLAMPED_WITHOUT_PART_ANALOG : Bool;   // UNIT 02 FIXTURE 3 PARTIAL UNCLAMPED
      UNCLAMPED_ANALOG : Bool;   // UNIT 02 FIXTURE 3 UNCLAMPED
      ALL_CNC_PLC_VARIABLES_ZERO : Bool;   // UNIT 02 FIXTURE 3 ALL CNC PLC VARIABLES ZERO
      FIXTURE_NOT_CLAMPED_ALARM : Bool;   // UNIT 02 FIXTURE 3 NOT CLAMPED DURING MACHINING ALARM
      PART_A_PRESENT_DISCORDANCY : Bool;   // UNIT 02 FIXTURE 3 PART A PRESENT DISCORDANCY
      PART_B_PRESENT_DISCORDANCY : Bool;   // UNIT 02 FIXTURE 3 PART B PRESENT DISCORDANCY
      PART_C_PRESENT_DISCORDANCY : Bool;   // UNIT 02 FIXTURE 3 PART C PRESENT DISCORDANCY
      PART_D_PRESENT_DISCORDANCY : Bool;   // UNIT 02 FIXTURE 3 PART D PRESENT DISCORDANCY
      PART_A_ORIENTATED_DISCORDANCY : Bool;   // UNIT 02 FIXTURE 3 PART A ORIENTATED DISCORDANCY
      PART_B_ORIENTATED_DISCORDANCY : Bool;   // UNIT 02 FIXTURE 3 PART B ORIENTATED DISCORDANCY
      PART_C_ORIENTATED_DISCORDANCY : Bool;   // UNIT 02 FIXTURE 3 PART C ORIENTATED DISCORDANCY
      PART_D_ORIENTATED_DISCORDANCY : Bool;   // UNIT 02 FIXTURE 3 PART D ORIENTATED DISCORDANCY
      PART_TYPE_DISCORDANCY : Bool;   // UNIT 02 FIXTURE 3 PART TYPE DISCORDANCY
      ANY_PART_PRESENT : Bool;   // UNIT 02 FIXTURE 3 ANY PART PRESENT
      CLAMPED_MEMORY_DONE : Bool;   // UNIT 02 FIXTURE 3 CLAMPED MEMORY DONE
      AUX_1 : Bool;
      AUX_2 : Bool;
      AUX_3 : Bool;
      TIMER_CLAMPED_DELAY : TON_TIME;   // UNIT 02 FIXTURE 3 CLAMPED TIMER
      TIMER_PART_A_ORIENTATION { S7_SetPoint := 'True'} : TON_TIME;   // UNIT 02 FIXTURE 3 PART A ORIENTATION TIMER
      TIMER_PART_A_DISCORDANCY { S7_SetPoint := 'True'} : TON_TIME;   // UNIT 02 FIXTURE 3 PART A DISCORDANCY TIMER
      TIMER_PART_C_ORIENTATION { S7_SetPoint := 'True'} : TON_TIME;   // UNIT 02 FIXTURE 3 PART C ORIENTATION TIMER
      TIMER_PART_D_ORIENTATION { S7_SetPoint := 'True'} : TON_TIME;   // UNIT 02 FIXTURE 3 PART D ORIENTATION TIMER
      TIMER_CLAMPED_WITH_ANALOG { S7_SetPoint := 'True'} : TOF_TIME;
   END_VAR
BEGIN
   TIMER_PART_A_ORIENTATION.PT := T#200ms;
   TIMER_PART_A_DISCORDANCY.PT := T#200ms;
   TIMER_PART_C_ORIENTATION.PT := T#200ms;
   TIMER_PART_D_ORIENTATION.PT := T#200ms;
   TIMER_CLAMPED_WITH_ANALOG.PT := T#100ms;
END_DATA_BLOCK

DATA_BLOCK "DB3800_UNIT_02_FIXTURE_4"   // DB3800
{ S7_Optimized_Access := 'FALSE'; DB_Accessible_From_OPC_UA := 'FALSE' }
AUTHOR : ETXETAR
VERSION : 1.0
// stored: AutoNumber false, DBAccessibleFromOPCUA false, DBAccessibleFromWebserver true, IsOnlyStoredInLoadMemory false, IsWriteProtectedInAS false
   VAR RETAIN
      INPUT_PART_A_PRESENT : Bool;   // UNIT 02 FIXTURE 4 INPUT PART A PRESENT
      INPUT_PART_B_PRESENT : Bool;   // UNIT 02 FIXTURE 4 INPUT PART B PRESENT
      INPUT_PART_C_PRESENT : Bool;   // UNIT 02 FIXTURE 4 INPUT PART C PRESENT
      INPUT_PART_D_PRESENT : Bool;   // UNIT 02 FIXTURE 4 INPUT PART D PRESENT
      INPUT_PART_A_PRESENT_FACE_N : Bool;   // UNIT 02 FIXTURE 4 INPUT PART A PRESENT FACE N UP
      INPUT_PART_B_PRESENT_FACE_N : Bool;   // UNIT 02 FIXTURE 4 INPUT PART B PRESENT FACE N UP
      INPUT_PART_C_PRESENT_FACE_N : Bool;   // UNIT 02 FIXTURE 4 INPUT PART C PRESENT FACE N UP
      INPUT_PART_D_PRESENT_FACE_N : Bool;   // UNIT 02 FIXTURE 4 INPUT PART D PRESENT FACE N UP
      INPUT_PART_A_PRESENT_FACE_R : Bool;   // UNIT 02 FIXTURE 4 INPUT PART A PRESENT FACE R UP
      INPUT_PART_B_PRESENT_FACE_R : Bool;   // UNIT 02 FIXTURE 4 INPUT PART B PRESENT FACE R UP
      INPUT_PART_C_PRESENT_FACE_R : Bool;   // UNIT 02 FIXTURE 4 INPUT PART C PRESENT FACE R UP
      INPUT_PART_D_PRESENT_FACE_R : Bool;   // UNIT 02 FIXTURE 4 INPUT PART D PRESENT FACE R UP
      INPUT_PART_A_PRESENT_MEM : Bool;   // UNIT 02 FIXTURE 4 INPUT PART A PRESENT MEMORY
      INPUT_PART_B_PRESENT_MEM : Bool;   // UNIT 02 FIXTURE 4 INPUT PART B PRESENT MEMORY
      INPUT_PART_C_PRESENT_MEM : Bool;   // UNIT 02 FIXTURE 4 INPUT PART C PRESENT MEMORY
      INPUT_PART_D_PRESENT_MEM : Bool;   // UNIT 02 FIXTURE 4 INPUT PART D PRESENT MEMORY
      INPUT_PART_A_PRESENT_FACE_N_MEM : Bool;   // UNIT 02 FIXTURE 4 INPUT PART A PRESENT FACE N UP MEMORY
      INPUT_PART_B_PRESENT_FACE_N_MEM : Bool;   // UNIT 02 FIXTURE 4 INPUT PART B PRESENT FACE N UP MEMORY
      INPUT_PART_C_PRESENT_FACE_N_MEM : Bool;   // UNIT 02 FIXTURE 4 INPUT PART C PRESENT FACE N UP MEMORY
      INPUT_PART_D_PRESENT_FACE_N_MEM : Bool;   // UNIT 02 FIXTURE 4 INPUT PART D PRESENT FACE N UP MEMORY
      INPUT_PART_A_PRESENT_FACE_R_MEM : Bool;   // UNIT 02 FIXTURE 4 INPUT PART A PRESENT FACE R UP MEMORY
      INPUT_PART_B_PRESENT_FACE_R_MEM : Bool;   // UNIT 02 FIXTURE 4 INPUT PART B PRESENT FACE R UP MEMORY
      INPUT_PART_C_PRESENT_FACE_R_MEM : Bool;   // UNIT 02 FIXTURE 4 INPUT PART C PRESENT FACE R UP MEMORY
      INPUT_PART_D_PRESENT_FACE_R_MEM : Bool;   // UNIT 02 FIXTURE 4 INPUT PART D PRESENT FACE R UP MEMORY
      CLAMPED_WITH_PART_A : Bool;   // UNIT 02 FIXTURE 4 CLAMPED WITH PART A
      CLAMPED_WITH_PART_B : Bool;   // UNIT 02 FIXTURE 4 CLAMPED WITH PART B
      CLAMPED_WITH_PART_C : Bool;   // UNIT 02 FIXTURE 4 CLAMPED WITH PART C
      CLAMPED_WITH_PART_D : Bool;   // UNIT 02 FIXTURE 4 CLAMPED WITH PART D
      CLAMPED_WITHOUT_PART_A : Bool;   // UNIT 02 FIXTURE 4 CLAMPED WITHOUT PART A
      CLAMPED_WITHOUT_PART_B : Bool;   // UNIT 02 FIXTURE 4 CLAMPED WITHOUT PART B
      CLAMPED_WITHOUT_PART_C : Bool;   // UNIT 02 FIXTURE 4 CLAMPED WITHOUT PART C
      CLAMPED_WITHOUT_PART_D : Bool;   // UNIT 02 FIXTURE 4 CLAMPED WITHOUT PART D
      CLAMPED_WITH_PARTS : Bool;   // UNIT 02 FIXTURE 4 CLAMPED WITH PARTS
      CLAMPED_WITHOUT_PARTS : Bool;   // UNIT 02 FIXTURE 4 CLAMPED WITHOUT PARTS
      PARTIAL_CLAMPED : Bool;   // UNIT 02 FIXTURE 4 PARTIAL CLAMPED
      CLAMPED_WITH_PART_ANALOG : Bool;   // UNIT 02 FIXTURE 4 CLAMPED
      CLAMPED_OK : Bool;   // UNIT 02 FIXTURE 4 CLAMPED OK
      CLAMPED_DELAYED : Bool;   // UNIT 02 FIXTURE 4 CLAMPED DELAYED
      CLAMPED_WITHOUT_PART_ANALOG : Bool;   // UNIT 02 FIXTURE 4 PARTIAL UNCLAMPED
      UNCLAMPED_ANALOG : Bool;   // UNIT 02 FIXTURE 4 UNCLAMPED
      ALL_CNC_PLC_VARIABLES_ZERO : Bool;   // UNIT 02 FIXTURE 4 ALL CNC PLC VARIABLES ZERO
      FIXTURE_NOT_CLAMPED_ALARM : Bool;   // UNIT 02 FIXTURE 4 NOT CLAMPED DURING MACHINING ALARM
      PART_A_PRESENT_DISCORDANCY : Bool;   // UNIT 02 FIXTURE 4 PART A PRESENT DISCORDANCY
      PART_B_PRESENT_DISCORDANCY : Bool;   // UNIT 02 FIXTURE 4 PART B PRESENT DISCORDANCY
      PART_C_PRESENT_DISCORDANCY : Bool;   // UNIT 02 FIXTURE 4 PART C PRESENT DISCORDANCY
      PART_D_PRESENT_DISCORDANCY : Bool;   // UNIT 02 FIXTURE 4 PART D PRESENT DISCORDANCY
      PART_A_ORIENTATED_DISCORDANCY : Bool;   // UNIT 02 FIXTURE 4 PART A ORIENTATED DISCORDANCY
      PART_B_ORIENTATED_DISCORDANCY : Bool;   // UNIT 02 FIXTURE 4 PART B ORIENTATED DISCORDANCY
      PART_C_ORIENTATED_DISCORDANCY : Bool;   // UNIT 02 FIXTURE 4 PART C ORIENTATED DISCORDANCY
      PART_D_ORIENTATED_DISCORDANCY : Bool;   // UNIT 02 FIXTURE 4 PART D ORIENTATED DISCORDANCY
      PART_TYPE_DISCORDANCY : Bool;   // UNIT 02 FIXTURE 4 PART TYPE DISCORDANCY
      ANY_PART_PRESENT : Bool;   // UNIT 02 FIXTURE 4 ANY PART PRESENT
      CLAMPED_MEMORY_DONE : Bool;   // UNIT 02 FIXTURE 4 CLAMPED MEMORY DONE
      AUX_1 : Bool;
      AUX_2 : Bool;
      AUX_3 : Bool;
      TIMER_CLAMPED_DELAY : TON_TIME;   // UNIT 02 FIXTURE 4 CLAMPED TIMER
      TIMER_PART_A_ORIENTATION { S7_SetPoint := 'True'} : TON_TIME;   // UNIT 02 FIXTURE 4 PART A ORIENTATION TIMER
      TIMER_PART_A_DISCORDANCY { S7_SetPoint := 'True'} : TON_TIME;   // UNIT 02 FIXTURE 4 PART A DISCORDANCY TIMER
      TIMER_PART_C_ORIENTATION { S7_SetPoint := 'True'} : TON_TIME;   // UNIT 02 FIXTURE 4 PART C ORIENTATION TIMER
      TIMER_PART_D_ORIENTATION { S7_SetPoint := 'True'} : TON_TIME;   // UNIT 02 FIXTURE 4 PART D ORIENTATION TIMER
      TIMER_CLAMPED_WITH_ANALOG { S7_SetPoint := 'True'} : TOF_TIME;
   END_VAR
BEGIN
   TIMER_PART_A_ORIENTATION.PT := T#200ms;
   TIMER_PART_A_DISCORDANCY.PT := T#200ms;
   TIMER_PART_C_ORIENTATION.PT := T#200ms;
   TIMER_PART_D_ORIENTATION.PT := T#200ms;
   TIMER_CLAMPED_WITH_ANALOG.PT := T#100ms;
END_DATA_BLOCK

DATA_BLOCK "DB4000_FIX_TABLE_POSITIONS"   // DB4000
{ S7_Optimized_Access := 'FALSE'; DB_Accessible_From_OPC_UA := 'FALSE' }
AUTHOR : ETXETAR
VERSION : 1.0
// stored: AutoNumber false, DBAccessibleFromOPCUA false, DBAccessibleFromWebserver true, IsOnlyStoredInLoadMemory false, IsWriteProtectedInAS false
   VAR RETAIN
      UNIT_01 : Struct
         FIXTURE_1 : Struct
            IN_LOAD_UNLOAD_STATION_1 : Bool;   // UNIT 01 FIXTURE 1 IN LOAD UNLOAD STATION
            IN_SPARE_STATION_2 : Bool;   // UNIT 01 FIXTURE 1 IN SPARE STATION
            IN_CLADDING_STATION_3 : Bool;   // UNIT 01 FIXTURE 1 IN CLADDING STATION
            IN_CLEAN_STATION_4 : Bool;   // UNIT 01 FIXTURE 1 IN CLEANING STATION
            NO_DEFINED_POSITION : Bool;   // UNIT 01 FIXTURE 1 IN NO DEFINED POSITION
         END_STRUCT;
         FIXTURE_2 : Struct
            IN_LOAD_UNLOAD_STATION_1 : Bool;   // UNIT 01 FIXTURE 2 IN LOAD UNLOAD STATION
            IN_SPARE_STATION_2 : Bool;   // UNIT 01 FIXTURE 2 IN SPARE STATION
            IN_CLADDING_STATION_3 : Bool;   // UNIT 01 FIXTURE 2 IN CLADDING STATION
            IN_CLEAN_STATION_4 : Bool;   // UNIT 01 FIXTURE 2 IN CLEANING STATION
            NO_DEFINED_POSITION : Bool;   // UNIT 01 FIXTURE 2 IN NO DEFINED POSITION
         END_STRUCT;
         FIXTURE_3 : Struct
            IN_LOAD_UNLOAD_STATION_1 : Bool;   // UNIT 01 FIXTURE 3 IN LOAD UNLOAD STATION
            IN_SPARE_STATION_2 : Bool;   // UNIT 01 FIXTURE 3 IN SPARE STATION
            IN_CLADDING_STATION_3 : Bool;   // UNIT 01 FIXTURE 3 IN CLADDING STATION
            IN_CLEAN_STATION_4 : Bool;   // UNIT 01 FIXTURE 3 IN CLEANING STATION
            NO_DEFINED_POSITION : Bool;   // UNIT 01 FIXTURE 3 IN NO DEFINED POSITION
         END_STRUCT;
         FIXTURE_4 : Struct
            IN_LOAD_UNLOAD_STATION_1 : Bool;   // UNIT 01 FIXTURE 4 IN LOAD UNLOAD STATION
            IN_SPARE_STATION_2 : Bool;   // UNIT 01 FIXTURE 4 IN SPARE STATION
            IN_CLADDING_STATION_3 : Bool;   // UNIT 01 FIXTURE 4 IN CLADDING STATION
            IN_CLEAN_STATION_4 : Bool;   // UNIT 01 FIXTURE 4 IN CLEANING STATION
            NO_DEFINED_POSITION : Bool;   // UNIT 01 FIXTURE 4 IN NO DEFINED POSITION
         END_STRUCT;
         AXIS_E10_HOME_POS : Bool;   // AXIS E10 IN HOME POSITION
         AXIS_E10_NOT_DEFINED_POS : Bool;   // AXIS E10 NOT IN A DEFINED POSITION
         SPARE : UInt;   // AXIS E10 POSITION SENSOR VALUE
         E10_POSITION_REACH : Struct
            E10_0_DEGREES : Bool;   // E10 AXIS 0 DEGREES POSITION REACH
            E10_90_DEGREES : Bool;   // E10 AXIS 90 DEGREES POSITION REACH
            E10_180_DEGREES : Bool;   // E10 AXIS 180 DEGREES POSITION REACH
            E10_270_DEGREES : Bool;   // E10 AXIS 270 DEGREES POSITION REACH
            E10_0_DEGREES_FLANGE : Bool;   // E10 AXIS 0 DEGREES POSITION REACH FLANGE
            E10_90_DEGREES_FLANGE : Bool;   // E10 AXIS 90 DEGREES POSITION REACH FLANGE
            E10_180_DEGREES_FLANGE : Bool;   // E10 AXIS 180 DEGREES POSITION REACH FLANGE
            E10_270_DEGREES_FLANGE : Bool;   // E10 AXIS 270 DEGREES POSITION REACH FLANGE
         END_STRUCT;
         FIXTURE_NUMBER_IN : Struct
            STATION_1 : Int;   // FIXTURE NUMBER IN STATION 1
            STATION_2 : Int;   // FIXTURE NUMBER IN STATION 2
            STATION_3 : Int;   // FIXTURE NUMBER IN STATION 3
            STATION_4 : Int;   // FIXTURE NUMBER IN STATION 4
         END_STRUCT;
      END_STRUCT;
      UNIT_02 : Struct
         FIXTURE_1 : Struct
            IN_LOAD_UNLOAD_STATION_1 : Bool;   // UNIT 02 FIXTURE 1 IN LOAD UNLOAD STATION
            IN_MEASURING_STATION_2 : Bool;   // UNIT 02 FIXTURE 1 IN SPARE STATION
            IN_CLADDING_STATION_3 : Bool;   // UNIT 02 FIXTURE 1 IN CLADDING STATION
            IN_CLEAN_STATION_4 : Bool;   // UNIT 02 FIXTURE 1 IN MEASURING/CLEANING STATION
            NO_DEFINED_POSITION : Bool;   // UNIT 02 FIXTURE 1 IN NO DEFINED POSITION
         END_STRUCT;
         FIXTURE_2 : Struct
            IN_LOAD_UNLOAD_STATION_1 : Bool;   // UNIT 02 FIXTURE 2 IN LOAD UNLOAD STATION
            IN_MEASURING_STATION_2 : Bool;   // UNIT 02 FIXTURE 2 IN SPARE STATION
            IN_CLADDING_STATION_3 : Bool;   // UNIT 02 FIXTURE 2 IN CLADDING STATION
            IN_CLEAN_STATION_4 : Bool;   // UNIT 02 FIXTURE 2 IN MEASURING/CLEANING STATION
            NO_DEFINED_POSITION : Bool;   // UNIT 02 FIXTURE 2 IN NO DEFINED POSITION
         END_STRUCT;
         FIXTURE_3 : Struct
            IN_LOAD_UNLOAD_STATION_1 : Bool;   // UNIT 02 FIXTURE 3 IN LOAD UNLOAD STATION
            IN_MEASURING_STATION_2 : Bool;   // UNIT 02 FIXTURE 3 IN SPARE STATION
            IN_CLADDING_STATION_3 : Bool;   // UNIT 02 FIXTURE 3 IN CLADDING STATION
            IN_CLEAN_STATION_4 : Bool;   // UNIT 02 FIXTURE 3 IN MEASURING/CLEANING STATION
            NO_DEFINED_POSITION : Bool;   // UNIT 02 FIXTURE 3 IN NO DEFINED POSITION
         END_STRUCT;
         FIXTURE_4 : Struct
            IN_LOAD_UNLOAD_STATION_1 : Bool;   // UNIT 02 FIXTURE 4 IN LOAD UNLOAD STATION
            IN_MEASURING_STATION_2 : Bool;   // UNIT 02 FIXTURE 4 IN SPARE STATION
            IN_CLADDING_STATION_3 : Bool;   // UNIT 02 FIXTURE 4 IN CLADDING STATION
            IN_CLEAN_STATION_4 : Bool;   // UNIT 02 FIXTURE 4 IN MEASURING/CLEANING STATION
            NO_DEFINED_POSITION : Bool;   // UNIT 02 FIXTURE 4 IN NO DEFINED POSITION
         END_STRUCT;
         AXIS_E20_HOME_POS : Bool;   // AXIS E20 IN HOME POSITION
         AXIS_E20_NOT_DEFINED_POS : Bool;   // AXIS E20 NOT IN A DEFINED POSITION
         SPARE : UInt;   // E20 POSITION SENSOR VALUE
         E20_POSITION_REACH : Struct
            E20_0_DEGREES : Bool;   // E20 AXIS 0 DEGREES POSITION REACH
            E20_90_DEGREES : Bool;   // E20 AXIS 90 DEGREES POSITION REACH
            E20_180_DEGREES : Bool;   // E20 AXIS 180 DEGREES POSITION REACH
            E20_270_DEGREES : Bool;   // E20 AXIS 270 DEGREES POSITION REACH
            E20_0_DEGREES_FLANGE : Bool;   // E20 AXIS 0 DEGREES POSITION REACH FLANGE
            E20_90_DEGREES_FLANGE : Bool;   // E20 AXIS 90 DEGREES POSITION REACH FLANGE
            E20_180_DEGREES_FLANGE : Bool;   // E20 AXIS 180 DEGREES POSITION REACH FLANGE
            E20_270_DEGREES_FLANGE : Bool;   // E20 AXIS 270 DEGREES POSITION REACH FLANGE
         END_STRUCT;
         FIXTURE_NUMBER_IN : Struct
            STATION_1 : Int;   // FIXTURE NUMBER IN STATION 1
            STATION_2 : Int;   // FIXTURE NUMBER IN STATION 2
            STATION_3 : Int;   // FIXTURE NUMBER IN STATION 3
            STATION_4 : Int;   // FIXTURE NUMBER IN STATION 4
         END_STRUCT;
      END_STRUCT;
   END_VAR
BEGIN
END_DATA_BLOCK

DATA_BLOCK "DB4001_FIXTURES_CALIBRATION"   // DB4001
{ S7_Optimized_Access := 'FALSE'; DB_Accessible_From_OPC_UA := 'FALSE' }
VERSION : 0.1
// stored: AutoNumber false, DBAccessibleFromOPCUA false, DBAccessibleFromWebserver true, IsOnlyStoredInLoadMemory false, IsWriteProtectedInAS false
   VAR
      FIXTURE_1_STA_2_CALIB_MEM : Bool;   // FIXTURE 1 STATION 2 CALIBRATION MEMORY
      FIXTURE_1_STA_3_CALIB_MEM : Bool;   // FIXTURE 1 STATION 3 CALIBRATION MEMORY
      FIXTURE_2_STA_2_CALIB_MEM : Bool;   // FIXTURE 2 STATION 2 CALIBRATION MEMORY
      FIXTURE_2_STA_3_CALIB_MEM : Bool;   // FIXTURE 2 STATION 3 CALIBRATION MEMORY
      FIXTURE_3_STA_2_CALIB_MEM : Bool;   // FIXTURE 3 STATION 2 CALIBRATION MEMORY
      FIXTURE_3_STA_3_CALIB_MEM : Bool;   // FIXTURE 3 STATION 3 CALIBRATION MEMORY
      FIXTURE_4_STA_2_CALIB_MEM : Bool;   // FIXTURE 4 STATION 2 CALIBRATION MEMORY
      FIXTURE_4_STA_3_CALIB_MEM : Bool;   // FIXTURE 4 STATION 3 CALIBRATION MEMORY
      ALL_FIXTURES_STA_2_CALIB_MEM : Bool;   // ALL FIXTURES STATION 2 CALIBRATION MEMORY
      ALL_FIXTURES_STA_3_CALIB_MEM : Bool;   // ALL FIXTURES STATION 3 CALIBRATION MEMORY
      ALL_FIXTURES_CALIB_MEM : Bool;   // ALL FIXTURES CALIBRATION MEMORY DONE
   END_VAR
BEGIN
END_DATA_BLOCK

DATA_BLOCK "DB6500_SMC_CYLINDER_HMI"   // DB6500
{ S7_Optimized_Access := 'FALSE'; DB_Accessible_From_OPC_UA := 'FALSE' }
VERSION : 0.1
// stored: AutoNumber false, DBAccessibleFromOPCUA false, DBAccessibleFromWebserver true, IsOnlyStoredInLoadMemory false, IsWriteProtectedInAS false
   VAR
      JXCP_AXIS_HMI_SELECTION : Word := 16#1;   // SELECTED AXIS FOR JXCP1 CONTROLLER
      JXCP_AXIS_MAIN_DB_HMI : Word;   // MAIN SIGNALS SELECTED JXCP1 CONTROLLER
      JXCP_AXIS_AUX_DB_HMI : Word;   // AUX SIGNALS SELECTED JXCP1 CONTROLLER
      LEC_AXIS_HMI_SELECTION : Word := 16#1;   // SELECTED AXIS FOR LECSN CONTROLLER
      LEC_AXIS_CONTROLLER_SIGNALS : Word;   // CONTROLLER SIGNALS
      LEC_AXIS_DATA : Word;   // AXIS DATA
   END_VAR
BEGIN
END_DATA_BLOCK

DATA_BLOCK "DB7001_UNIT_01_MAIN_SAFETY_DOOR"   // DB7001
{ S7_Optimized_Access := 'FALSE'; DB_Accessible_From_OPC_UA := 'FALSE' }
AUTHOR : ETXETAR
VERSION : 1.0
// stored: AutoNumber false, DBAccessibleFromOPCUA false, DBAccessibleFromWebserver true, IsOnlyStoredInLoadMemory false, IsWriteProtectedInAS false
   VAR RETAIN
      SAFETY_DOOR : "SAFETY_DOOR";
   END_VAR
BEGIN
   SAFETY_DOOR.TIMER_PARTIAL_UNLOCK_GENERAL_CONDITIONS.PT := T#60ms;
   SAFETY_DOOR.TIMER_UNLOCK.PT := T#500ms;
   SAFETY_DOOR.TIMER_NOT_POSSIBLE_TO_UNLOCK.PT := T#1s;
END_DATA_BLOCK

DATA_BLOCK "DB7002_UNIT_01_STATION_02_SAFETY_DOOR"   // DB7002
{ S7_Optimized_Access := 'FALSE'; DB_Accessible_From_OPC_UA := 'FALSE' }
AUTHOR : ETXETAR
VERSION : 1.0
// stored: AutoNumber false, DBAccessibleFromOPCUA false, DBAccessibleFromWebserver true, IsOnlyStoredInLoadMemory false, IsWriteProtectedInAS false
   VAR RETAIN
      SAFETY_DOOR : "SAFETY_DOOR";
   END_VAR
BEGIN
   SAFETY_DOOR.TIMER_PARTIAL_UNLOCK_GENERAL_CONDITIONS.PT := T#60ms;
   SAFETY_DOOR.TIMER_UNLOCK.PT := T#500ms;
   SAFETY_DOOR.TIMER_NOT_POSSIBLE_TO_UNLOCK.PT := T#1s;
END_DATA_BLOCK

DATA_BLOCK "DB7003_UNIT_01_STATION_04_SAFETY_DOOR"   // DB7003
{ S7_Optimized_Access := 'FALSE'; DB_Accessible_From_OPC_UA := 'FALSE' }
AUTHOR : ETXETAR
VERSION : 1.0
// stored: AutoNumber false, DBAccessibleFromOPCUA false, DBAccessibleFromWebserver true, IsOnlyStoredInLoadMemory false, IsWriteProtectedInAS false
   VAR RETAIN
      SAFETY_DOOR : "SAFETY_DOOR";
   END_VAR
BEGIN
   SAFETY_DOOR.TIMER_PARTIAL_UNLOCK_GENERAL_CONDITIONS.PT := T#60ms;
   SAFETY_DOOR.TIMER_UNLOCK.PT := T#500ms;
   SAFETY_DOOR.TIMER_NOT_POSSIBLE_TO_UNLOCK.PT := T#1s;
END_DATA_BLOCK

DATA_BLOCK "DB7011_UNIT_02_MAIN_SAFETY_DOOR"   // DB7011
{ S7_Optimized_Access := 'FALSE'; DB_Accessible_From_OPC_UA := 'FALSE' }
AUTHOR : ETXETAR
VERSION : 1.0
// stored: AutoNumber false, DBAccessibleFromOPCUA false, DBAccessibleFromWebserver true, IsOnlyStoredInLoadMemory false, IsWriteProtectedInAS false
   VAR RETAIN
      SAFETY_DOOR : "SAFETY_DOOR";
   END_VAR
BEGIN
   SAFETY_DOOR.TIMER_PARTIAL_UNLOCK_GENERAL_CONDITIONS.PT := T#500ms;
   SAFETY_DOOR.TIMER_UNLOCK.PT := T#500ms;
   SAFETY_DOOR.TIMER_NOT_POSSIBLE_TO_UNLOCK.PT := T#1s;
END_DATA_BLOCK

DATA_BLOCK "DB7012_UNIT_02_STATION_02_SAFETY_DOOR"   // DB7012
{ S7_Optimized_Access := 'FALSE'; DB_Accessible_From_OPC_UA := 'FALSE' }
AUTHOR : ETXETAR
VERSION : 1.0
// stored: AutoNumber false, DBAccessibleFromOPCUA false, DBAccessibleFromWebserver true, IsOnlyStoredInLoadMemory false, IsWriteProtectedInAS false
   VAR RETAIN
      SAFETY_DOOR : "SAFETY_DOOR";
   END_VAR
BEGIN
   SAFETY_DOOR.TIMER_PARTIAL_UNLOCK_GENERAL_CONDITIONS.PT := T#60ms;
   SAFETY_DOOR.TIMER_UNLOCK.PT := T#500ms;
   SAFETY_DOOR.TIMER_NOT_POSSIBLE_TO_UNLOCK.PT := T#1s;
END_DATA_BLOCK

DATA_BLOCK "DB7013_UNIT_02_STATION_04_SAFETY_DOOR"   // DB7013
{ S7_Optimized_Access := 'FALSE'; DB_Accessible_From_OPC_UA := 'FALSE' }
AUTHOR : ETXETAR
VERSION : 1.0
// stored: AutoNumber false, DBAccessibleFromOPCUA false, DBAccessibleFromWebserver true, IsOnlyStoredInLoadMemory false, IsWriteProtectedInAS false
   VAR RETAIN
      SAFETY_DOOR : "SAFETY_DOOR";
   END_VAR
BEGIN
   SAFETY_DOOR.TIMER_PARTIAL_UNLOCK_GENERAL_CONDITIONS.PT := T#500ms;
   SAFETY_DOOR.TIMER_UNLOCK.PT := T#500ms;
   SAFETY_DOOR.TIMER_NOT_POSSIBLE_TO_UNLOCK.PT := T#1s;
END_DATA_BLOCK

DATA_BLOCK "DB7200_HMI_FUNCTION"   // DB7200
{ S7_Optimized_Access := 'FALSE'; DB_Accessible_From_OPC_UA := 'FALSE' }
AUTHOR : ETXETAR
VERSION : 1.0
// stored: AutoNumber false, DBAccessibleFromOPCUA false, DBAccessibleFromWebserver true, IsOnlyStoredInLoadMemory false, IsWriteProtectedInAS false
   VAR RETAIN
      HELP_PROMPT : Int;   // HELP PROMPT
      PLC_SCREEN_SELECTION : Word;   // PLC SCREEN SELECTION
      SCREEN_SELECTION : Array[11..89] of Bool;   // SCREEN SELECTION
   END_VAR
BEGIN
END_DATA_BLOCK

DATA_BLOCK "DB8001_UNIT_01_PART_STATUS_HMI"   // DB8001
{ S7_Optimized_Access := 'FALSE'; DB_Accessible_From_OPC_UA := 'FALSE' }
VERSION : 0.1
// stored: AutoNumber false, DBAccessibleFromOPCUA false, DBAccessibleFromWebserver true, IsOnlyStoredInLoadMemory false, IsWriteProtectedInAS false
   VAR
      Int_PART_TYPE : Array[0..63] of Char;
      WChar_PART_TYPE : Array[0..63] of WChar;
   END_VAR
BEGIN
END_DATA_BLOCK

DATA_BLOCK "DB8002_UNIT_02_PART_STATUS_HMI"   // DB8002
{ S7_Optimized_Access := 'FALSE'; DB_Accessible_From_OPC_UA := 'FALSE' }
VERSION : 0.1
// stored: AutoNumber false, DBAccessibleFromOPCUA false, DBAccessibleFromWebserver true, IsOnlyStoredInLoadMemory false, IsWriteProtectedInAS false
   VAR
      Int_PART_TYPE : Array[0..63] of Char;
      WChar_PART_TYPE : Array[0..63] of WChar;
   END_VAR
BEGIN
END_DATA_BLOCK

DATA_BLOCK "DB8100_MANUAL_LOADING_PART_STATUS"   // DB8100
{ S7_Optimized_Access := 'FALSE'; DB_Accessible_From_OPC_UA := 'FALSE' }
VERSION : 0.1
// stored: AutoNumber false, DBAccessibleFromOPCUA false, DBAccessibleFromWebserver true, IsOnlyStoredInLoadMemory false, IsWriteProtectedInAS false
   VAR
      UNIT_01_DELETE_PART_HMI_BUTTON : Bool;   // DELETE PART FROM FIXTURE IN UNIT 01 STATION 1 HMI BUTTON
      UNIT_01_ADD_PART_HMI_BUTTON : Bool;   // ADD PART TO FIXTURE IN UNIT 01 STATION 1 HMI BUTTON
      UNIT_01_SKIP_LOADING_FIX_STA_1_HMI_BUTTON : Bool;   // UNIT 01 SKIP LOADING FIXTURE IN STATION 1 HMI BUTTON
      UNIT_01_NO_FACE_R_PARTS_TO_DELIVER : Bool;   // NO FACE R PARTS TO DELIVER UNIT 01
      UNIT_01_NO_FACE_N_PARTS_TO_DELIVER : Bool;   // NO FACE N PARTS TO DELIVER UNIT 01
      UNIT_01_SPARE_3 : Bool;
      UNIT_01_SPARE_4 : Bool;
      UNIT_01_SPARE_5 : Bool;
      UNIT_02_DELETE_PART_HMI_BUTTON : Bool;   // DELETE PART FROM FIXTURE IN UNIT 02 STATION 1 HMI BUTTON
      UNIT_02_ADD_PART_HMI_BUTTON : Bool;   // ADD PART TO FIXTURE IN UNIT 02 STATION 1 HMI BUTTON
      UNIT_02_SKIP_LOADING_FIX_STA_1_HMI_BUTTON : Bool;   // UNIT 02 SKIP LOADING FIXTURE IN STATION 1 HMI BUTTON
      UNIT_02_NO_FACE_R_PARTS_TO_DELIVER : Bool;   // NO FACE R PARTS TO DELIVER UNIT 02
      UNIT_02_NO_FACE_N_PARTS_TO_DELIVER : Bool;   // NO FACE N PARTS TO DELIVER UNIT 02
      UNIT_02_SPARE_3 : Bool;
      UNIT_02_SPARE_4 : Bool;
      UNIT_02_SPARE_5 : Bool;
      UNIT_03_DELETE_PART_HMI_BUTTON : Bool;   // DELETE PART FROM FIXTURE IN UNIT 03 STATION 1 HMI BUTTON
      UNIT_03_ADD_PART_HMI_BUTTON : Bool;   // ADD PART TO FIXTURE IN UNIT 03 STATION 1 HMI BUTTON
      UNIT_03_SPARE_1 : Bool;
      UNIT_03_SPARE_2 : Bool;
      UNIT_03_SPARE_3 : Bool;
      UNIT_03_SPARE_4 : Bool;
      UNIT_03_SPARE_5 : Bool;
      UNIT_03_SPARE_6 : Bool;
   END_VAR
BEGIN
END_DATA_BLOCK

ORGANIZATION_BLOCK "OB1_CYCLE"   // OB1, LAD, ProgramCycle
TITLE = "Main Program Sweep (Cycle)"
{ S7_Optimized_Access := 'FALSE' }
VERSION : 0.1
// stored: AutoNumber false, IsIECCheckEnabled false, SetENOAutomatically false
   VAR_TEMP
      EV_CLASS : Byte;   // Bits 0-3 = 1:Coming event, Bits 4-7 = 1:Event class 1
      SCAN_1 : Byte;   // 1:Initial call of the OB, 3: Call 2-n of the OB
      PRIORITY : Byte;   // Priority of OB Execution
      OB_NUMBR : Byte;   // OB number
      RESERVED_1 : Byte;   // Reserved for system
      RESERVED_2 : Byte;   // Reserved for system
      PREV_CYCLE : Int;   // Previous program cycle time (milliseconds)
      MIN_CYCLE : Int;   // Minimum program cycle time (milliseconds)
      MAX_CYCLE : Int;   // Maximum program cycle time (milliseconds)
      DATE_TIME : Date_And_Time;   // Date and time OB started
      OB1_SCAN : Byte;   // 1 (Cold restart scan 1 of OB 1), 3 (Scan 2-n of OB 1)
      OB1_PRIORITY : Int;   // Priority of OB Execution
      OB1_MIN_CYCLE : DInt;   // Minimum cycle time of OB1 (milliseconds)
      OB1_MAX_CYCLE : DInt;   // Maximum cycle time of OB1 (milliseconds)
      PART_TYPE : Int;
      zero : Byte;
      status_sfc21 : Int;
      Error : Bool;
      status : Word;
   END_VAR
   VAR_TEMP   // added for the SCL form of the ladder/FBD networks
      _w1 : Bool;
   END_VAR
BEGIN

REGION Network 1: M ZERO - M ONE
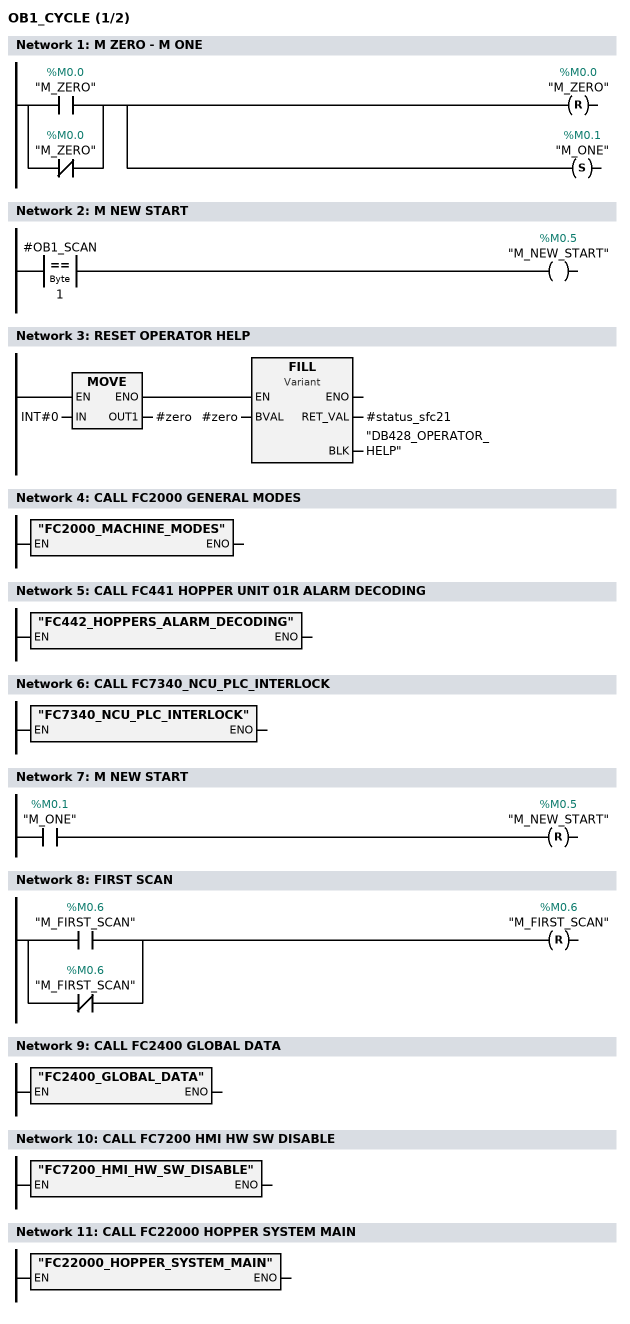
   RUNG wire#powerrail
      Contact( "M_ZERO" )
      wire#w1
      R_Coil( "M_ZERO" )
   END_RUNG
   RUNG wire#powerrail
      I_Contact( "M_ZERO" )
   END_RUNG wire#w1
   RUNG wire#w1
      S_Coil( "M_ONE" )
   END_RUNG
   // the same network as SCL:
   #_w1 := "M_ZERO" OR NOT "M_ZERO";
   IF #_w1 THEN
       "M_ZERO" := FALSE;
       "M_ONE" := TRUE;
   END_IF;
END_REGION

REGION Network 2: M NEW START
   RUNG wire#powerrail
      { S7_Templates := "SrcType := Byte" } EQ_Contact(in1 := #OB1_SCAN, in2 := 1)
      Coil( "M_NEW_START" )
   END_RUNG
   // the same network as SCL:
   "M_NEW_START" := #OB1_SCAN = 1;
END_REGION

REGION Network 3: RESET OPERATOR HELP
   RUNG wire#powerrail
      { S7_GenerateENO := "TRUE" } Move(in := INT#0, out1 => #zero)
      { S7_Templates := "ptr_type := Variant" } FILL(BVAL := #zero, RET_VAL => #status_sfc21, BLK => "DB428_OPERATOR_HELP")
   END_RUNG
   // the same network as SCL:
   // ENO of a box is taken as its EN; it also drops when the box reports an error
   #zero := INT#0;
   #status_sfc21 := FILL(BVAL := #zero, BLK => "DB428_OPERATOR_HELP");
END_REGION

REGION Network 4: CALL FC2000 GENERAL MODES
   RUNG wire#powerrail
      "FC2000_MACHINE_MODES"()
   END_RUNG
   // the same network as SCL:
   "FC2000_MACHINE_MODES"();
END_REGION

REGION Network 5: CALL FC441 HOPPER UNIT 01R ALARM DECODING
   RUNG wire#powerrail
      "FC442_HOPPERS_ALARM_DECODING"()
   END_RUNG
   // the same network as SCL:
   "FC442_HOPPERS_ALARM_DECODING"();
END_REGION

REGION Network 6: CALL FC7340_NCU_PLC_INTERLOCK
   RUNG wire#powerrail
      "FC7340_NCU_PLC_INTERLOCK"()
   END_RUNG
   // the same network as SCL:
   "FC7340_NCU_PLC_INTERLOCK"();
END_REGION

REGION Network 7: M NEW START
   RUNG wire#powerrail
      Contact( "M_ONE" )
      R_Coil( "M_NEW_START" )
   END_RUNG
   // the same network as SCL:
   IF "M_ONE" THEN "M_NEW_START" := FALSE; END_IF;
END_REGION

REGION Network 8: FIRST SCAN
   RUNG wire#powerrail
      Contact( "M_FIRST_SCAN" )
      wire#w1
      R_Coil( "M_FIRST_SCAN" )
   END_RUNG
   RUNG wire#powerrail
      I_Contact( "M_FIRST_SCAN" )
   END_RUNG wire#w1
   // the same network as SCL:
   IF "M_FIRST_SCAN" OR NOT "M_FIRST_SCAN" THEN "M_FIRST_SCAN" := FALSE; END_IF;
END_REGION

REGION Network 9: CALL FC2400 GLOBAL DATA
   RUNG wire#powerrail
      "FC2400_GLOBAL_DATA"()
   END_RUNG
   // the same network as SCL:
   "FC2400_GLOBAL_DATA"();
END_REGION

REGION Network 10: CALL FC7200 HMI HW SW DISABLE
   RUNG wire#powerrail
      "FC7200_HMI_HW_SW_DISABLE"()
   END_RUNG
   // the same network as SCL:
   "FC7200_HMI_HW_SW_DISABLE"();
END_REGION

REGION Network 11: CALL FC22000 HOPPER SYSTEM MAIN
   RUNG wire#powerrail
      "FC22000_HOPPER_SYSTEM_MAIN"()
   END_RUNG
   // the same network as SCL:
   "FC22000_HOPPER_SYSTEM_MAIN"();
END_REGION

REGION Network 12: CALL FC2100 GENERAL
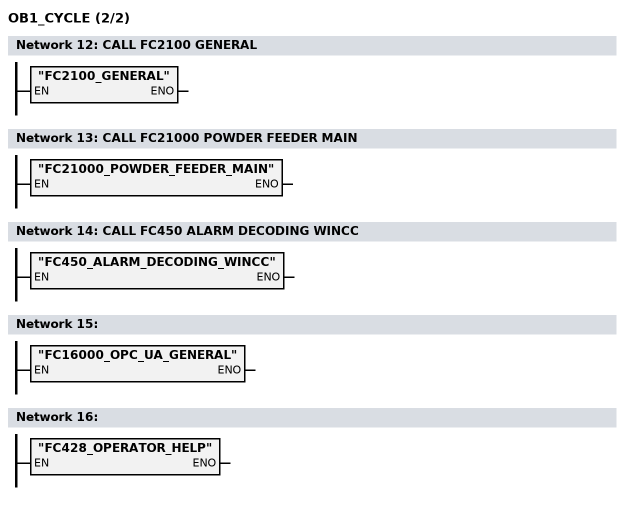
   RUNG wire#powerrail
      "FC2100_GENERAL"()
   END_RUNG
   // the same network as SCL:
   "FC2100_GENERAL"();
END_REGION

REGION Network 13: CALL FC21000 POWDER FEEDER MAIN
   RUNG wire#powerrail
      "FC21000_POWDER_FEEDER_MAIN"()
   END_RUNG
   // the same network as SCL:
   "FC21000_POWDER_FEEDER_MAIN"();
END_REGION

REGION Network 14: CALL FC450 ALARM DECODING WINCC
   RUNG wire#powerrail
      "FC450_ALARM_DECODING_WINCC"()
   END_RUNG
   // the same network as SCL:
   "FC450_ALARM_DECODING_WINCC"();
END_REGION

REGION Network 15
   RUNG wire#powerrail
      "FC16000_OPC_UA_GENERAL"()
   END_RUNG
   // the same network as SCL:
   "FC16000_OPC_UA_GENERAL"();
END_REGION

REGION Network 16
   RUNG wire#powerrail
      "FC428_OPERATOR_HELP"()
   END_RUNG
   // the same network as SCL:
   "FC428_OPERATOR_HELP"();
END_REGION
END_ORGANIZATION_BLOCK

FUNCTION "FC2000_MACHINE_MODES" : Void   // FC2000, LAD
{ S7_Optimized_Access := 'FALSE' }
AUTHOR : ETXETAR
VERSION : 1.0
// stored: AutoNumber false, IsIECCheckEnabled false, SetENOAutomatically false, UDAEnableTagReadback false
BEGIN

REGION Network 1: OPTIONS OFF
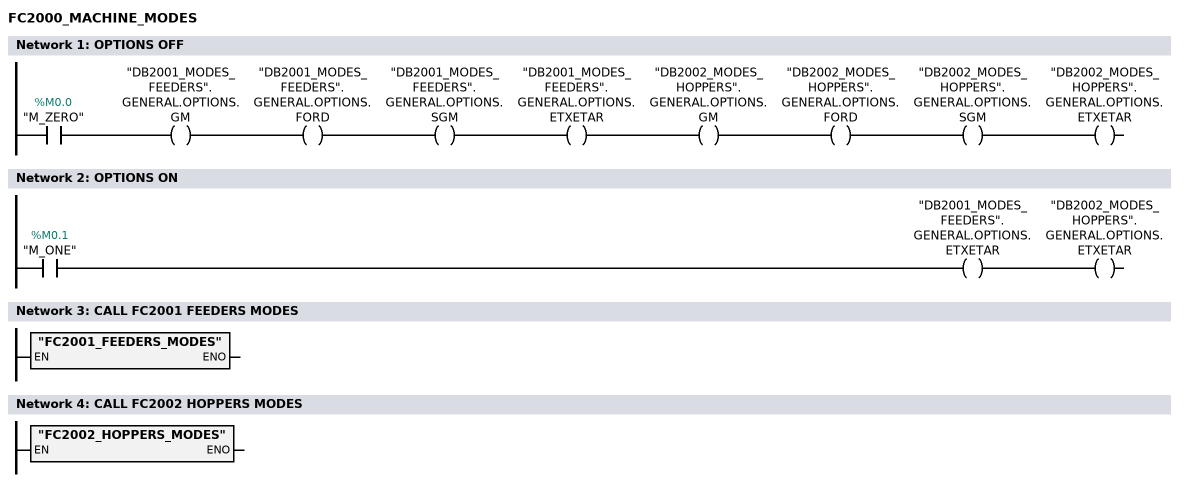
   RUNG wire#powerrail
      Contact( "M_ZERO" )
      Coil( "DB2001_MODES_FEEDERS".GENERAL.OPTIONS.GM )
      Coil( "DB2001_MODES_FEEDERS".GENERAL.OPTIONS.FORD )
      Coil( "DB2001_MODES_FEEDERS".GENERAL.OPTIONS.SGM )
      Coil( "DB2001_MODES_FEEDERS".GENERAL.OPTIONS.ETXETAR )
      Coil( "DB2002_MODES_HOPPERS".GENERAL.OPTIONS.GM )
      Coil( "DB2002_MODES_HOPPERS".GENERAL.OPTIONS.FORD )
      Coil( "DB2002_MODES_HOPPERS".GENERAL.OPTIONS.SGM )
      Coil( "DB2002_MODES_HOPPERS".GENERAL.OPTIONS.ETXETAR )
   END_RUNG
   // the same network as SCL:
   "DB2001_MODES_FEEDERS".GENERAL.OPTIONS.GM := "M_ZERO";
   "DB2001_MODES_FEEDERS".GENERAL.OPTIONS.FORD := "M_ZERO";
   "DB2001_MODES_FEEDERS".GENERAL.OPTIONS.SGM := "M_ZERO";
   "DB2001_MODES_FEEDERS".GENERAL.OPTIONS.ETXETAR := "M_ZERO";
   "DB2002_MODES_HOPPERS".GENERAL.OPTIONS.GM := "M_ZERO";
   "DB2002_MODES_HOPPERS".GENERAL.OPTIONS.FORD := "M_ZERO";
   "DB2002_MODES_HOPPERS".GENERAL.OPTIONS.SGM := "M_ZERO";
   "DB2002_MODES_HOPPERS".GENERAL.OPTIONS.ETXETAR := "M_ZERO";
END_REGION

REGION Network 2: OPTIONS ON
   RUNG wire#powerrail
      Contact( "M_ONE" )
      Coil( "DB2001_MODES_FEEDERS".GENERAL.OPTIONS.ETXETAR )
      Coil( "DB2002_MODES_HOPPERS".GENERAL.OPTIONS.ETXETAR )
   END_RUNG
   // the same network as SCL:
   "DB2001_MODES_FEEDERS".GENERAL.OPTIONS.ETXETAR := "M_ONE";
   "DB2002_MODES_HOPPERS".GENERAL.OPTIONS.ETXETAR := "M_ONE";
END_REGION

REGION Network 3: CALL FC2001 FEEDERS MODES
   RUNG wire#powerrail
      "FC2001_FEEDERS_MODES"()
   END_RUNG
   // the same network as SCL:
   "FC2001_FEEDERS_MODES"();
END_REGION

REGION Network 4: CALL FC2002 HOPPERS MODES
   RUNG wire#powerrail
      "FC2002_HOPPERS_MODES"()
   END_RUNG
   // the same network as SCL:
   "FC2002_HOPPERS_MODES"();
END_REGION
END_FUNCTION

FUNCTION "FC7200_HMI_HW_SW_DISABLE" : Void   // FC7200, LAD
{ S7_Optimized_Access := 'TRUE' }
VERSION : 0.1
// stored: AutoNumber false, IsIECCheckEnabled false, SetENOAutomatically false, UDAEnableTagReadback false
BEGIN

REGION Network 1: CALL FC7238 VARIABLES PLC CONNECTION
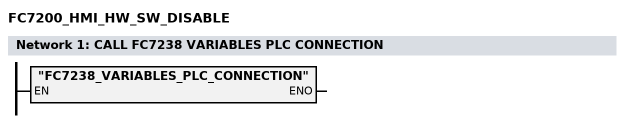
   RUNG wire#powerrail
      "FC7238_VARIABLES_PLC_CONNECTION"()
   END_RUNG
   // the same network as SCL:
   "FC7238_VARIABLES_PLC_CONNECTION"();
END_REGION
END_FUNCTION

FUNCTION "FC22000_HOPPER_SYSTEM_MAIN" : Void   // FC22000, LAD
TITLE = FC22000 HOPPER SYSTEM MAIN
{ S7_Optimized_Access := 'TRUE' }
VERSION : 0.1
// stored: AutoNumber false, IsIECCheckEnabled false, SetENOAutomatically false, UDAEnableTagReadback false
BEGIN

REGION Network 1: FC22100_HOPPER_SYSTEM_SENSORS
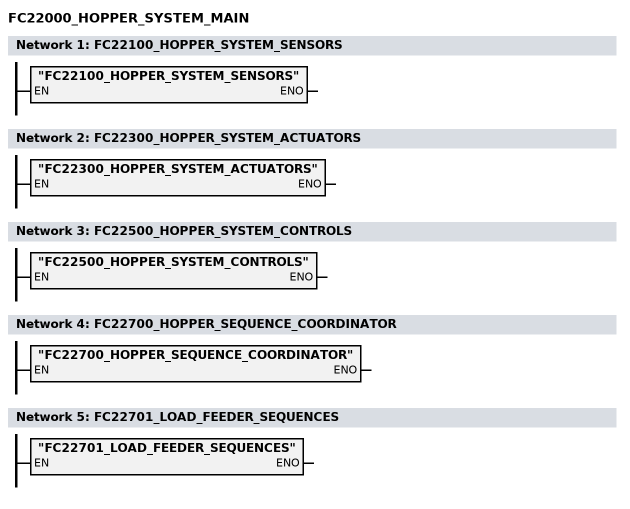
   RUNG wire#powerrail
      "FC22100_HOPPER_SYSTEM_SENSORS"()
   END_RUNG
   // the same network as SCL:
   "FC22100_HOPPER_SYSTEM_SENSORS"();
END_REGION

REGION Network 2: FC22300_HOPPER_SYSTEM_ACTUATORS
   RUNG wire#powerrail
      "FC22300_HOPPER_SYSTEM_ACTUATORS"()
   END_RUNG
   // the same network as SCL:
   "FC22300_HOPPER_SYSTEM_ACTUATORS"();
END_REGION

REGION Network 3: FC22500_HOPPER_SYSTEM_CONTROLS
   RUNG wire#powerrail
      "FC22500_HOPPER_SYSTEM_CONTROLS"()
   END_RUNG
   // the same network as SCL:
   "FC22500_HOPPER_SYSTEM_CONTROLS"();
END_REGION

REGION Network 4: FC22700_HOPPER_SEQUENCE_COORDINATOR
   RUNG wire#powerrail
      "FC22700_HOPPER_SEQUENCE_COORDINATOR"()
   END_RUNG
   // the same network as SCL:
   "FC22700_HOPPER_SEQUENCE_COORDINATOR"();
END_REGION

REGION Network 5: FC22701_LOAD_FEEDER_SEQUENCES
   RUNG wire#powerrail
      "FC22701_LOAD_FEEDER_SEQUENCES"()
   END_RUNG
   // the same network as SCL:
   "FC22701_LOAD_FEEDER_SEQUENCES"();
END_REGION
END_FUNCTION

FUNCTION "FC22100_HOPPER_SYSTEM_SENSORS" : Void   // FC22100, LAD
TITLE = FC22100 HOPPER SYSTEM SENSORS
{ S7_Optimized_Access := 'TRUE' }
VERSION : 0.1
// stored: AutoNumber false, IsIECCheckEnabled false, SetENOAutomatically false, UDAEnableTagReadback false
   VAR CONSTANT
      FC_NUMBER : UInt := 22100;
   END_VAR
   VAR_TEMP   // added for the SCL form of the ladder/FBD networks
      _w1 : Bool;
   END_VAR
BEGIN

REGION Network 1: /////_UNIT_01_SENSORS_/////
END_REGION

